LIN {X 0,Y 522.426,Z 691.44,A -85,B 0,C 180,E1 4711.435,E2 4711.435} C_VEL
LIN {X 0,Y 522.387,Z 691.44,A -85,B 0,C 180,E1 4717.482,E2 4717.482} C_VEL
LIN {X 0,Y 522.255,Z 691.44,A -85,B 0,C 180,E1 4723.549,E2 4723.549} C_VEL
LIN {X 0,Y 522.445,Z 691.44,A -85,B 0,C 180,E1 4730.119,E2 4730.119} C_VEL
LIN {X 0,Y 522.544,Z 692.414,A -85,B 0,C 180,E1 4730.325,E2 4730.325} C_VEL
LIN {X 0,Y 539.275,Z 726.671,A -85,B 0,C 180,E1 4732.514,E2 4732.514} C_VEL
LIN {X 0,Y 537.589,Z 764.271,A -85,B 0,C 180,E1 4733.74,E2 4733.74} C_VEL
LIN {X 0,Y 535.249,Z 801.949,A -85,B 0,C 180,E1 4735.545,E2 4735.545} C_VEL
LIN {X 0,Y 532.435,Z 840.351,A -85,B 0,C 180,E1 4738.098,E2 4738.098} C_VEL
LIN {X 0,Y 529.459,Z 877.291,A -85,B 0,C 180,E1 4741.38,E2 4741.38} C_VEL
LIN {X 0,Y 526.999,Z 909.325,A -85,B 0,C 180,E1 4745.105,E2 4745.105} C_VEL
LIN {X 0,Y 525.112,Z 937.42,A -85,B 0,C 180,E1 4749.358,E2 4749.358} C_VEL
LIN {X 0,Y 523.97,Z 958.909,A -85,B 0,C 180,E1 4753.636,E2 4753.636} C_VEL
LIN {X 0,Y 523.391,Z 974.577,A -85,B 0,C 180,E1 4757.893,E2 4757.893} C_VEL
LIN {X 0,Y 523.168,Z 984.427,A -85,B 0,C 180,E1 4761.68,E2 4761.68} C_VEL
LIN {X 0,Y 523.113,Z 989.961,A -85,B 0,C 180,E1 4765.018,E2 4765.018} C_VEL
LIN {X 0,Y 523.072,Z 992.674,A -85,B 0,C 180,E1 4768.341,E2 4768.341} C_VEL
LIN {X 0,Y 523.125,Z 992.634,A -85,B 0,C 180,E1 4771.658,E2 4771.658} C_VEL
LIN {X 0,Y 523.173,Z 988.638,A -85,B 0,C 180,E1 4775.813,E2 4775.813} C_VEL
LIN {X 0,Y 523.346,Z 980.316,A -85,B 0,C 180,E1 4779.996,E2 4779.996} C_VEL
LIN {X 0,Y 523.726,Z 965.346,A -85,B 0,C 180,E1 4784.698,E2 4784.698} C_VEL
LIN {X 0,Y 524.624,Z 945.078,A -85,B 0,C 180,E1 4789.164,E2 4789.164} C_VEL
LIN {X 0,Y 526.306,Z 918.749,A -85,B 0,C 180,E1 4793.507,E2 4793.507} C_VEL
LIN {X 0,Y 528.671,Z 887.696,A -85,B 0,C 180,E1 4797.423,E2 4797.423} C_VEL
LIN {X 0,Y 531.474,Z 852.279,A -85,B 0,C 180,E1 4800.85,E2 4800.85} C_VEL
LIN {X 0,Y 534.394,Z 814.101,A -85,B 0,C 180,E1 4803.642,E2 4803.642} C_VEL
LIN {X 0,Y 537.05,Z 773.839,A -85,B 0,C 180,E1 4805.776,E2 4805.776} C_VEL
LIN {X 0,Y 539,Z 734.912,A -85,B 0,C 180,E1 4807.168,E2 4807.168} C_VEL
LIN {X 0,Y 538.832,Z 725.059,A -85,B 0,C 180,E1 4807.474,E2 4807.474} C_VEL
LIN {X 0,Y 522.37,Z 692.689,A -85,B 0,C 180,E1 4809.596,E2 4809.596} C_VEL
LIN {X 0,Y 522.274,Z 691.44,A -85,B 0,C 180,E1 4809.626,E2 4809.626} C_VEL
LIN {X 0,Y 522.4,Z 691.44,A -85,B 0,C 180,E1 4815.938,E2 4815.938} C_VEL
LIN {X 0,Y 522.319,Z 691.44,A -85,B 0,C 180,E1 4821.505,E2 4821.505} C_VEL
LIN {X 0,Y 522.347,Z 691.44,A -85,B 0,C 180,E1 4827.203,E2 4827.203} C_VEL
LIN {X 0,Y 522.46,Z 691.44,A -85,B 0,C 180,E1 4832.384,E2 4832.384} C_VEL
LIN {X 0,Y 522.611,Z 691.44,A -85,B 0,C 180,E1 4837.985,E2 4837.985} C_VEL
LIN {X 0,Y 522.696,Z 691.44,A -85,B 0,C 180,E1 4843.169,E2 4843.169} C_VEL
LIN {X 0,Y 522.745,Z 691.44,A -85,B 0,C 180,E1 4848.308,E2 4848.308} C_VEL
LIN {X 0,Y 522.774,Z 691.44,A -85,B 0,C 180,E1 4853.352,E2 4853.352} C_VEL
LIN {X 0,Y 522.845,Z 691.44,A -85,B 0,C 180,E1 4858.345,E2 4858.345} C_VEL
LIN {X 0,Y 522.824,Z 691.44,A -85,B 0,C 180,E1 4863.324,E2 4863.324} C_VEL
LIN {X 0,Y 522.696,Z 691.44,A -85,B 0,C 180,E1 4868.331,E2 4868.331} C_VEL
LIN {X 0,Y 522.66,Z 691.44,A -85,B 0,C 180,E1 4873.402,E2 4873.402} C_VEL
LIN {X 0,Y 522.58,Z 691.44,A -85,B 0,C 180,E1 4878.586,E2 4878.586} C_VEL
LIN {X 0,Y 522.567,Z 691.44,A -85,B 0,C 180,E1 4883.932,E2 4883.932} C_VEL
LIN {X 0,Y 522.359,Z 691.44,A -85,B 0,C 180,E1 4889.593,E2 4889.593} C_VEL
LIN {X 0,Y 522.321,Z 691.44,A -85,B 0,C 180,E1 4892.498,E2 4892.498} C_VEL
LIN {X 0,Y 519.868,Z 691.44,A -85,B 0,C 180,E1 4893.912,E2 4893.912} C_VEL
LIN {X 0,Y 514.507,Z 691.44,A -85,B 0,C 180,E1 4896.031,E2 4896.031} C_VEL
LIN {X 0,Y 514.405,Z 691.44,A -85,B 0,C 180,E1 4896.276,E2 4896.276} C_VEL
LIN {X 0,Y 514.452,Z 691.44,A -85,B 0,C 180,E1 4902.601,E2 4902.601} C_VEL
LIN {X 0,Y 514.39,Z 691.44,A -85,B 0,C 180,E1 4909.063,E2 4909.063} C_VEL
LIN {X 0,Y 516.656,Z 696.972,A -85,B 0,C 180,E1 4909.378,E2 4909.378} C_VEL
LIN {X 0,Y 533.601,Z 728.662,A -85,B 0,C 180,E1 4911.452,E2 4911.452} C_VEL
LIN {X 0,Y 532.248,Z 772.885,A -85,B 0,C 180,E1 4912.494,E2 4912.494} C_VEL
LIN {X 0,Y 529.856,Z 813.695,A -85,B 0,C 180,E1 4914.129,E2 4914.129} C_VEL
LIN {X 0,Y 526.866,Z 853.448,A -85,B 0,C 180,E1 4916.444,E2 4916.444} C_VEL
LIN {X 0,Y 523.9,Z 889.133,A -85,B 0,C 180,E1 4919.257,E2 4919.257} C_VEL
LIN {X 0,Y 521.019,Z 921.486,A -85,B 0,C 180,E1 4922.555,E2 4922.555} C_VEL
LIN {X 0,Y 518.699,Z 950.198,A -85,B 0,C 180,E1 4926.305,E2 4926.305} C_VEL
LIN {X 0,Y 516.878,Z 975.351,A -85,B 0,C 180,E1 4930.546,E2 4930.546} C_VEL
LIN {X 0,Y 515.909,Z 995.049,A -85,B 0,C 180,E1 4934.952,E2 4934.952} C_VEL
LIN {X 0,Y 515.398,Z 1009.438,A -85,B 0,C 180,E1 4939.475,E2 4939.475} C_VEL
LIN {X 0,Y 515.274,Z 1017.479,A -85,B 0,C 180,E1 4943.25,E2 4943.25} C_VEL
LIN {X 0,Y 515.21,Z 1022.223,A -85,B 0,C 180,E1 4947.588,E2 4947.588} C_VEL
LIN {X 0,Y 515.151,Z 1022.657,A -85,B 0,C 180,E1 4951.685,E2 4951.685} C_VEL
LIN {X 0,Y 515.278,Z 1018.703,A -85,B 0,C 180,E1 4955.903,E2 4955.903} C_VEL
LIN {X 0,Y 515.502,Z 1010.436,A -85,B 0,C 180,E1 4960.15,E2 4960.15} C_VEL
LIN {X 0,Y 515.962,Z 995.944,A -85,B 0,C 180,E1 4964.803,E2 4964.803} C_VEL
LIN {X 0,Y 516.915,Z 975.395,A -85,B 0,C 180,E1 4969.443,E2 4969.443} C_VEL
LIN {X 0,Y 518.818,Z 949.033,A -85,B 0,C 180,E1 4973.869,E2 4973.869} C_VEL
LIN {X 0,Y 521.438,Z 917.371,A -85,B 0,C 180,E1 4977.919,E2 4977.919} C_VEL
LIN {X 0,Y 524.469,Z 882.798,A -85,B 0,C 180,E1 4981.308,E2 4981.308} C_VEL
LIN {X 0,Y 527.597,Z 844.909,A -85,B 0,C 180,E1 4984.124,E2 4984.124} C_VEL
LIN {X 0,Y 530.493,Z 804.797,A -85,B 0,C 180,E1 4986.284,E2 4986.284} C_VEL
LIN {X 0,Y 532.713,Z 762.573,A -85,B 0,C 180,E1 4987.804,E2 4987.804} C_VEL
LIN {X 0,Y 533.345,Z 728.122,A -85,B 0,C 180,E1 4988.579,E2 4988.579} C_VEL
LIN {X 0,Y 514.534,Z 692.798,A -85,B 0,C 180,E1 4990.898,E2 4990.898} C_VEL
LIN {X 0,Y 514.426,Z 691.44,A -85,B 0,C 180,E1 4991.055,E2 4991.055} C_VEL
LIN {X 0,Y 514.439,Z 691.44,A -85,B 0,C 180,E1 4997.398,E2 4997.398} C_VEL
LIN {X 0,Y 514.454,Z 691.44,A -85,B 0,C 180,E1 5002.621,E2 5002.621} C_VEL
LIN {X 0,Y 514.454,Z 691.44,A -85,B 0,C 180,E1 5008.595,E2 5008.595} C_VEL
LIN {X 0,Y 514.559,Z 691.44,A -85,B 0,C 180,E1 5013.808,E2 5013.808} C_VEL
LIN {X 0,Y 514.675,Z 691.44,A -85,B 0,C 180,E1 5019.327,E2 5019.327} C_VEL
LIN {X 0,Y 514.565,Z 691.44,A -85,B 0,C 180,E1 5024.642,E2 5024.642} C_VEL
LIN {X 0,Y 514.737,Z 691.44,A -85,B 0,C 180,E1 5029.832,E2 5029.832} C_VEL
LIN {X 0,Y 514.959,Z 691.44,A -85,B 0,C 180,E1 5034.936,E2 5034.936} C_VEL
LIN {X 0,Y 515.019,Z 691.44,A -85,B 0,C 180,E1 5039.996,E2 5039.996} C_VEL
LIN {X 0,Y 514.944,Z 691.44,A -85,B 0,C 180,E1 5045.056,E2 5045.056} C_VEL
LIN {X 0,Y 514.872,Z 691.44,A -85,B 0,C 180,E1 5050.157,E2 5050.157} C_VEL
LIN {X 0,Y 514.778,Z 691.44,A -85,B 0,C 180,E1 5055.343,E2 5055.343} C_VEL
LIN {X 0,Y 514.675,Z 691.44,A -85,B 0,C 180,E1 5060.665,E2 5060.665} C_VEL
LIN {X 0,Y 514.55,Z 691.44,A -85,B 0,C 180,E1 5066.184,E2 5066.184} C_VEL
LIN {X 0,Y 514.549,Z 691.44,A -85,B 0,C 180,E1 5071.973,E2 5071.973} C_VEL
LIN {X 0,Y 514.472,Z 691.44,A -85,B 0,C 180,E1 5078.161,E2 5078.161} C_VEL
LIN {X 0,Y 514.337,Z 691.44,A -85,B 0,C 180,E1 5082.613,E2 5082.613} C_VEL
LIN {X 0,Y 514.486,Z 691.44,A -85,B 0,C 180,E1 5089.553,E2 5089.553} C_VEL
LIN {X 0,Y 518.78,Z 700.928,A -85,B 0,C 180,E1 5090.135,E2 5090.135} C_VEL
LIN {X 0,Y 532.868,Z 728.329,A -85,B 0,C 180,E1 5092.028,E2 5092.028} C_VEL
LIN {X 0,Y 530.904,Z 768.275,A -85,B 0,C 180,E1 5093.392,E2 5093.392} C_VEL
LIN {X 0,Y 528.322,Z 805.367,A -85,B 0,C 180,E1 5095.254,E2 5095.254} C_VEL
LIN {X 0,Y 525.28,Z 843.001,A -85,B 0,C 180,E1 5097.842,E2 5097.842} C_VEL
LIN {X 0,Y 522.172,Z 878.329,A -85,B 0,C 180,E1 5101.061,E2 5101.061} C_VEL
LIN {X 0,Y 519.593,Z 909.281,A -85,B 0,C 180,E1 5104.719,E2 5104.719} C_VEL
LIN {X 0,Y 517.486,Z 937.186,A -85,B 0,C 180,E1 5108.997,E2 5108.997} C_VEL
LIN {X 0,Y 516.17,Z 958.905,A -85,B 0,C 180,E1 5113.381,E2 5113.381} C_VEL
LIN {X 0,Y 515.535,Z 974.574,A -85,B 0,C 180,E1 5117.706,E2 5117.706} C_VEL
LIN {X 0,Y 515.281,Z 984.426,A -85,B 0,C 180,E1 5121.551,E2 5121.551} C_VEL
LIN {X 0,Y 515.228,Z 989.96,A -85,B 0,C 180,E1 5124.942,E2 5124.942} C_VEL
LIN {X 0,Y 515.171,Z 992.674,A -85,B 0,C 180,E1 5128.316,E2 5128.316} C_VEL
LIN {X 0,Y 515.143,Z 992.185,A -85,B 0,C 180,E1 5132.429,E2 5132.429} C_VEL
LIN {X 0,Y 515.253,Z 987.399,A -85,B 0,C 180,E1 5136.75,E2 5136.75} C_VEL
LIN {X 0,Y 515.468,Z 977.399,A -85,B 0,C 180,E1 5141.237,E2 5141.237} C_VEL
LIN {X 0,Y 515.923,Z 963.805,A -85,B 0,C 180,E1 5145.315,E2 5145.315} C_VEL
LIN {X 0,Y 516.943,Z 943.977,A -85,B 0,C 180,E1 5149.679,E2 5149.679} C_VEL
LIN {X 0,Y 518.796,Z 918.754,A -85,B 0,C 180,E1 5153.869,E2 5153.869} C_VEL
LIN {X 0,Y 521.415,Z 887.703,A -85,B 0,C 180,E1 5157.838,E2 5157.838} C_VEL
LIN {X 0,Y 524.471,Z 852.291,A -85,B 0,C 180,E1 5161.308,E2 5161.308} C_VEL
LIN {X 0,Y 527.69,Z 813.795,A -85,B 0,C 180,E1 5164.149,E2 5164.149} C_VEL
LIN {X 0,Y 530.577,Z 773.856,A -85,B 0,C 180,E1 5166.282,E2 5166.282} C_VEL
LIN {X 0,Y 532.746,Z 734.504,A -85,B 0,C 180,E1 5167.693,E2 5167.693} C_VEL
LIN {X 0,Y 532.192,Z 727.448,A -85,B 0,C 180,E1 5167.962,E2 5167.962} C_VEL
LIN {X 0,Y 514.479,Z 692.831,A -85,B 0,C 180,E1 5170.331,E2 5170.331} C_VEL
LIN {X 0,Y 514.347,Z 691.44,A -85,B 0,C 180,E1 5170.542,E2 5170.542} C_VEL
LIN {X 0,Y 514.415,Z 691.44,A -85,B 0,C 180,E1 5175.071,E2 5175.071} C_VEL
LIN {X 0,Y 514.472,Z 691.44,A -85,B 0,C 180,E1 5179.922,E2 5179.922} C_VEL
LIN {X 0,Y 514.359,Z 691.44,A -85,B 0,C 180,E1 5186.004,E2 5186.004} C_VEL
LIN {X 0,Y 514.501,Z 691.44,A -85,B 0,C 180,E1 5191.987,E2 5191.987} C_VEL
LIN {X 0,Y 514.647,Z 691.44,A -85,B 0,C 180,E1 5197.522,E2 5197.522} C_VEL
LIN {X 0,Y 514.776,Z 691.44,A -85,B 0,C 180,E1 5202.902,E2 5202.902} C_VEL
LIN {X 0,Y 514.832,Z 691.44,A -85,B 0,C 180,E1 5208.126,E2 5208.126} C_VEL
LIN {X 0,Y 514.864,Z 691.44,A -85,B 0,C 180,E1 5213.25,E2 5213.25} C_VEL
LIN {X 0,Y 514.956,Z 691.44,A -85,B 0,C 180,E1 5218.526,E2 5218.526} C_VEL
LIN {X 0,Y 514.92,Z 691.44,A -85,B 0,C 180,E1 5223.375,E2 5223.375} C_VEL
LIN {X 0,Y 514.782,Z 691.44,A -85,B 0,C 180,E1 5228.46,E2 5228.46} C_VEL
LIN {X 0,Y 514.733,Z 691.44,A -85,B 0,C 180,E1 5233.907,E2 5233.907} C_VEL
LIN {X 0,Y 514.621,Z 691.44,A -85,B 0,C 180,E1 5239.699,E2 5239.699} C_VEL
LIN {X 0,Y 514.641,Z 691.44,A -85,B 0,C 180,E1 5244.324,E2 5244.324} C_VEL
LIN {X 0,Y 514.421,Z 691.44,A -85,B 0,C 180,E1 5250.024,E2 5250.024} C_VEL
LIN {X 0,Y 514.405,Z 691.44,A -85,B 0,C 180,E1 5256.276,E2 5256.276} C_VEL
LIN {X 0,Y 513.115,Z 691.44,A -85,B 0,C 180,E1 5257.239,E2 5257.239} C_VEL
LIN {X 0,Y 506.485,Z 691.44,A -85,B 0,C 180,E1 5259.86,E2 5259.86} C_VEL
LIN {X 0,Y 506.394,Z 691.44,A -85,B 0,C 180,E1 5260.108,E2 5260.108} C_VEL
LIN {X 0,Y 506.412,Z 691.44,A -85,B 0,C 180,E1 5265.851,E2 5265.851} C_VEL
LIN {X 0,Y 506.521,Z 691.58,A -85,B 0,C 180,E1 5268.297,E2 5268.297} C_VEL
LIN {X 0,Y 510.766,Z 700.951,A -85,B 0,C 180,E1 5268.886,E2 5268.886} C_VEL
LIN {X 0,Y 527.479,Z 731.737,A -85,B 0,C 180,E1 5270.981,E2 5270.981} C_VEL
LIN {X 0,Y 525.902,Z 773.975,A -85,B 0,C 180,E1 5272,E2 5272} C_VEL
LIN {X 0,Y 523.228,Z 816.041,A -85,B 0,C 180,E1 5273.727,E2 5273.727} C_VEL
LIN {X 0,Y 519.776,Z 857.497,A -85,B 0,C 180,E1 5276.226,E2 5276.226} C_VEL
LIN {X 0,Y 516.312,Z 895.403,A -85,B 0,C 180,E1 5279.368,E2 5279.368} C_VEL
LIN {X 0,Y 513.008,Z 929.647,A -85,B 0,C 180,E1 5283.115,E2 5283.115} C_VEL
LIN {X 0,Y 510.483,Z 959.035,A -85,B 0,C 180,E1 5287.321,E2 5287.321} C_VEL
LIN {X 0,Y 508.819,Z 982.147,A -85,B 0,C 180,E1 5291.635,E2 5291.635} C_VEL
LIN {X 0,Y 507.923,Z 1000.301,A -85,B 0,C 180,E1 5296.204,E2 5296.204} C_VEL
LIN {X 0,Y 507.526,Z 1012.606,A -85,B 0,C 180,E1 5300.646,E2 5300.646} C_VEL
LIN {X 0,Y 507.424,Z 1019.905,A -85,B 0,C 180,E1 5304.865,E2 5304.865} C_VEL
LIN {X 0,Y 507.396,Z 1022.657,A -85,B 0,C 180,E1 5308.29,E2 5308.29} C_VEL
LIN {X 0,Y 507.319,Z 1021.627,A -85,B 0,C 180,E1 5313.422,E2 5313.422} C_VEL
LIN {X 0,Y 507.443,Z 1015.917,A -85,B 0,C 180,E1 5317.717,E2 5317.717} C_VEL
LIN {X 0,Y 507.636,Z 1005.771,A -85,B 0,C 180,E1 5322.051,E2 5322.051} C_VEL
LIN {X 0,Y 508.318,Z 990.49,A -85,B 0,C 180,E1 5326.438,E2 5326.438} C_VEL
LIN {X 0,Y 509.72,Z 969.378,A -85,B 0,C 180,E1 5330.883,E2 5330.883} C_VEL
LIN {X 0,Y 511.785,Z 943.259,A -85,B 0,C 180,E1 5335.069,E2 5335.069} C_VEL
LIN {X 0,Y 514.543,Z 913.188,A -85,B 0,C 180,E1 5338.806,E2 5338.806} C_VEL
LIN {X 0,Y 517.862,Z 878.743,A -85,B 0,C 180,E1 5342.117,E2 5342.117} C_VEL
LIN {X 0,Y 521.115,Z 842.642,A -85,B 0,C 180,E1 5344.764,E2 5344.764} C_VEL
LIN {X 0,Y 524.261,Z 802.755,A -85,B 0,C 180,E1 5346.894,E2 5346.894} C_VEL
LIN {X 0,Y 526.437,Z 762.992,A -85,B 0,C 180,E1 5348.322,E2 5348.322} C_VEL
LIN {X 0,Y 526.991,Z 730.718,A -85,B 0,C 180,E1 5349.082,E2 5349.082} C_VEL
LIN {X 0,Y 506.659,Z 692.982,A -85,B 0,C 180,E1 5351.664,E2 5351.664} C_VEL
LIN {X 0,Y 506.519,Z 691.44,A -85,B 0,C 180,E1 5351.811,E2 5351.811} C_VEL
LIN {X 0,Y 506.485,Z 691.44,A -85,B 0,C 180,E1 5358.362,E2 5358.362} C_VEL
LIN {X 0,Y 506.537,Z 691.44,A -85,B 0,C 180,E1 5363.81,E2 5363.81} C_VEL
LIN {X 0,Y 506.517,Z 691.44,A -85,B 0,C 180,E1 5370.098,E2 5370.098} C_VEL
LIN {X 0,Y 506.639,Z 691.44,A -85,B 0,C 180,E1 5375.266,E2 5375.266} C_VEL
LIN {X 0,Y 506.813,Z 691.44,A -85,B 0,C 180,E1 5380.813,E2 5380.813} C_VEL
LIN {X 0,Y 506.617,Z 691.44,A -85,B 0,C 180,E1 5386.165,E2 5386.165} C_VEL
LIN {X 0,Y 506.849,Z 691.44,A -85,B 0,C 180,E1 5391.407,E2 5391.407} C_VEL
LIN {X 0,Y 507.02,Z 691.44,A -85,B 0,C 180,E1 5396.572,E2 5396.572} C_VEL
LIN {X 0,Y 507.072,Z 691.44,A -85,B 0,C 180,E1 5401.707,E2 5401.707} C_VEL
LIN {X 0,Y 506.955,Z 691.44,A -85,B 0,C 180,E1 5406.856,E2 5406.856} C_VEL
LIN {X 0,Y 506.856,Z 691.44,A -85,B 0,C 180,E1 5412.064,E2 5412.064} C_VEL
LIN {X 0,Y 506.807,Z 691.44,A -85,B 0,C 180,E1 5417.376,E2 5417.376} C_VEL
LIN {X 0,Y 506.713,Z 691.44,A -85,B 0,C 180,E1 5422.85,E2 5422.85} C_VEL
LIN {X 0,Y 506.544,Z 691.44,A -85,B 0,C 180,E1 5428.562,E2 5428.562} C_VEL
LIN {X 0,Y 506.601,Z 691.44,A -85,B 0,C 180,E1 5434.59,E2 5434.59} C_VEL
LIN {X 0,Y 506.421,Z 691.44,A -85,B 0,C 180,E1 5441.116,E2 5441.116} C_VEL
LIN {X 0,Y 506.374,Z 691.44,A -85,B 0,C 180,E1 5446.55,E2 5446.55} C_VEL
LIN {X 0,Y 506.584,Z 691.44,A -85,B 0,C 180,E1 5448.757,E2 5448.757} C_VEL
LIN {X 0,Y 511.353,Z 701.712,A -85,B 0,C 180,E1 5449.447,E2 5449.447} C_VEL
LIN {X 0,Y 526.49,Z 731.264,A -85,B 0,C 180,E1 5451.58,E2 5451.58} C_VEL
LIN {X 0,Y 524.243,Z 772.496,A -85,B 0,C 180,E1 5453.047,E2 5453.047} C_VEL
LIN {X 0,Y 521.209,Z 811.429,A -85,B 0,C 180,E1 5455.116,E2 5455.116} C_VEL
LIN {X 0,Y 517.884,Z 848.298,A -85,B 0,C 180,E1 5457.8,E2 5457.8} C_VEL
LIN {X 0,Y 514.557,Z 882.537,A -85,B 0,C 180,E1 5461.076,E2 5461.076} C_VEL
LIN {X 0,Y 511.836,Z 912.444,A -85,B 0,C 180,E1 5464.77,E2 5464.77} C_VEL
LIN {X 0,Y 509.755,Z 938.401,A -85,B 0,C 180,E1 5468.891,E2 5468.891} C_VEL
LIN {X 0,Y 508.391,Z 958.902,A -85,B 0,C 180,E1 5473.119,E2 5473.119} C_VEL
LIN {X 0,Y 507.692,Z 974.571,A -85,B 0,C 180,E1 5477.513,E2 5477.513} C_VEL
LIN {X 0,Y 507.391,Z 984.424,A -85,B 0,C 180,E1 5481.419,E2 5481.419} C_VEL
LIN {X 0,Y 507.331,Z 989.959,A -85,B 0,C 180,E1 5484.863,E2 5484.863} C_VEL
LIN {X 0,Y 507.291,Z 992.674,A -85,B 0,C 180,E1 5488.289,E2 5488.289} C_VEL
LIN {X 0,Y 507.334,Z 992.635,A -85,B 0,C 180,E1 5491.71,E2 5491.71} C_VEL
LIN {X 0,Y 507.375,Z 988.64,A -85,B 0,C 180,E1 5495.995,E2 5495.995} C_VEL
LIN {X 0,Y 507.59,Z 979.171,A -85,B 0,C 180,E1 5500.744,E2 5500.744} C_VEL
LIN {X 0,Y 508.044,Z 965.517,A -85,B 0,C 180,E1 5505.116,E2 5505.116} C_VEL
LIN {X 0,Y 509.156,Z 945.376,A -85,B 0,C 180,E1 5509.711,E2 5509.711} C_VEL
LIN {X 0,Y 511.113,Z 920.579,A -85,B 0,C 180,E1 5513.963,E2 5513.963} C_VEL
LIN {X 0,Y 513.822,Z 890.873,A -85,B 0,C 180,E1 5517.894,E2 5517.894} C_VEL
LIN {X 0,Y 517.003,Z 857.416,A -85,B 0,C 180,E1 5521.32,E2 5521.32} C_VEL
LIN {X 0,Y 520.294,Z 822.156,A -85,B 0,C 180,E1 5524.088,E2 5524.088} C_VEL
LIN {X 0,Y 523.368,Z 783.668,A -85,B 0,C 180,E1 5526.343,E2 5526.343} C_VEL
LIN {X 0,Y 526.016,Z 743.231,A -85,B 0,C 180,E1 5527.972,E2 5527.972} C_VEL
LIN {X 0,Y 526.121,Z 731.045,A -85,B 0,C 180,E1 5528.369,E2 5528.369} C_VEL
LIN {X 0,Y 506.531,Z 692.262,A -85,B 0,C 180,E1 5531.117,E2 5531.117} C_VEL
LIN {X 0,Y 506.507,Z 691.44,A -85,B 0,C 180,E1 5531.657,E2 5531.657} C_VEL
LIN {X 0,Y 506.483,Z 691.44,A -85,B 0,C 180,E1 5538.361,E2 5538.361} C_VEL
LIN {X 0,Y 506.5,Z 691.44,A -85,B 0,C 180,E1 5543.814,E2 5543.814} C_VEL
LIN {X 0,Y 506.528,Z 691.44,A -85,B 0,C 180,E1 5550.094,E2 5550.094} C_VEL
LIN {X 0,Y 506.677,Z 691.44,A -85,B 0,C 180,E1 5555.277,E2 5555.277} C_VEL
LIN {X 0,Y 506.822,Z 691.44,A -85,B 0,C 180,E1 5560.822,E2 5560.822} C_VEL
LIN {X 0,Y 506.985,Z 691.44,A -85,B 0,C 180,E1 5566.184,E2 5566.184} C_VEL
LIN {X 0,Y 507.008,Z 691.44,A -85,B 0,C 180,E1 5571.418,E2 5571.418} C_VEL
LIN {X 0,Y 507.178,Z 691.44,A -85,B 0,C 180,E1 5576.582,E2 5576.582} C_VEL
LIN {X 0,Y 507.295,Z 691.44,A -85,B 0,C 180,E1 5581.714,E2 5581.714} C_VEL
LIN {X 0,Y 507.062,Z 691.44,A -85,B 0,C 180,E1 5586.863,E2 5586.863} C_VEL
LIN {X 0,Y 506.869,Z 691.44,A -85,B 0,C 180,E1 5592.072,E2 5592.072} C_VEL
LIN {X 0,Y 506.779,Z 691.44,A -85,B 0,C 180,E1 5597.385,E2 5597.385} C_VEL
LIN {X 0,Y 506.729,Z 691.44,A -85,B 0,C 180,E1 5602.858,E2 5602.858} C_VEL
LIN {X 0,Y 506.529,Z 691.44,A -85,B 0,C 180,E1 5608.572,E2 5608.572} C_VEL
LIN {X 0,Y 506.47,Z 691.44,A -85,B 0,C 180,E1 5614.611,E2 5614.611} C_VEL
LIN {X 0,Y 506.394,Z 691.44,A -85,B 0,C 180,E1 5620.108,E2 5620.108} C_VEL
LIN {X 0,Y 503.895,Z 691.44,A -85,B 0,C 180,E1 5621.569,E2 5621.569} C_VEL
LIN {X 0,Y 498.621,Z 691.44,A -85,B 0,C 180,E1 5623.758,E2 5623.758} C_VEL
LIN {X 0,Y 498.534,Z 691.44,A -85,B 0,C 180,E1 5624.011,E2 5624.011} C_VEL
LIN {X 0,Y 498.582,Z 691.44,A -85,B 0,C 180,E1 5627.457,E2 5627.457} C_VEL
LIN {X 0,Y 503.054,Z 701.159,A -85,B 0,C 180,E1 5628.126,E2 5628.126} C_VEL
LIN {X 0,Y 521.229,Z 734.453,A -85,B 0,C 180,E1 5630.479,E2 5630.479} C_VEL
LIN {X 0,Y 519.57,Z 775.534,A -85,B 0,C 180,E1 5631.516,E2 5631.516} C_VEL
LIN {X 0,Y 516.672,Z 817.16,A -85,B 0,C 180,E1 5633.256,E2 5633.256} C_VEL
LIN {X 0,Y 512.985,Z 858.207,A -85,B 0,C 180,E1 5635.775,E2 5635.775} C_VEL
LIN {X 0,Y 509.262,Z 895.435,A -85,B 0,C 180,E1 5638.901,E2 5638.901} C_VEL
LIN {X 0,Y 505.79,Z 928.839,A -85,B 0,C 180,E1 5642.589,E2 5642.589} C_VEL
LIN {X 0,Y 502.862,Z 959.037,A -85,B 0,C 180,E1 5646.957,E2 5646.957} C_VEL
LIN {X 0,Y 501.01,Z 983.299,A -85,B 0,C 180,E1 5651.605,E2 5651.605} C_VEL
LIN {X 0,Y 500.042,Z 1001.746,A -85,B 0,C 180,E1 5656.429,E2 5656.429} C_VEL
LIN {X 0,Y 499.556,Z 1014.331,A -85,B 0,C 180,E1 5661.284,E2 5661.284} C_VEL
LIN {X 0,Y 499.53,Z 1019.905,A -85,B 0,C 180,E1 5664.783,E2 5664.783} C_VEL
LIN {X 0,Y 499.5,Z 1022.657,A -85,B 0,C 180,E1 5668.263,E2 5668.263} C_VEL
LIN {X 0,Y 499.413,Z 1021.627,A -85,B 0,C 180,E1 5673.477,E2 5673.477} C_VEL
LIN {X 0,Y 499.554,Z 1015.917,A -85,B 0,C 180,E1 5677.839,E2 5677.839} C_VEL
LIN {X 0,Y 499.774,Z 1005.77,A -85,B 0,C 180,E1 5682.244,E2 5682.244} C_VEL
LIN {X 0,Y 500.541,Z 990.491,A -85,B 0,C 180,E1 5686.701,E2 5686.701} C_VEL
LIN {X 0,Y 502.073,Z 969.379,A -85,B 0,C 180,E1 5691.216,E2 5691.216} C_VEL
LIN {X 0,Y 504.382,Z 943.018,A -85,B 0,C 180,E1 5695.498,E2 5695.498} C_VEL
LIN {X 0,Y 507.324,Z 913.665,A -85,B 0,C 180,E1 5699.199,E2 5699.199} C_VEL
LIN {X 0,Y 510.819,Z 880.199,A -85,B 0,C 180,E1 5702.482,E2 5702.482} C_VEL
LIN {X 0,Y 514.483,Z 842.657,A -85,B 0,C 180,E1 5705.278,E2 5705.278} C_VEL
LIN {X 0,Y 517.913,Z 802.357,A -85,B 0,C 180,E1 5707.443,E2 5707.443} C_VEL
LIN {X 0,Y 520.361,Z 761.523,A -85,B 0,C 180,E1 5708.902,E2 5708.902} C_VEL
LIN {X 0,Y 520.917,Z 733.875,A -85,B 0,C 180,E1 5709.561,E2 5709.561} C_VEL
LIN {X 0,Y 498.647,Z 692.273,A -85,B 0,C 180,E1 5712.494,E2 5712.494} C_VEL
LIN {X 0,Y 498.552,Z 691.44,A -85,B 0,C 180,E1 5713.21,E2 5713.21} C_VEL
LIN {X 0,Y 498.514,Z 691.44,A -85,B 0,C 180,E1 5719.403,E2 5719.403} C_VEL
LIN {X 0,Y 498.573,Z 691.44,A -85,B 0,C 180,E1 5725.08,E2 5725.08} C_VEL
LIN {X 0,Y 498.583,Z 691.44,A -85,B 0,C 180,E1 5731.723,E2 5731.723} C_VEL
LIN {X 0,Y 498.759,Z 691.44,A -85,B 0,C 180,E1 5736.755,E2 5736.755} C_VEL
LIN {X 0,Y 498.876,Z 691.44,A -85,B 0,C 180,E1 5742.33,E2 5742.33} C_VEL
LIN {X 0,Y 498.771,Z 691.44,A -85,B 0,C 180,E1 5747.729,E2 5747.729} C_VEL
LIN {X 0,Y 499.133,Z 691.44,A -85,B 0,C 180,E1 5753.027,E2 5753.027} C_VEL
LIN {X 0,Y 499.38,Z 691.44,A -85,B 0,C 180,E1 5758.259,E2 5758.259} C_VEL
LIN {X 0,Y 499.259,Z 691.44,A -85,B 0,C 180,E1 5763.473,E2 5763.473} C_VEL
LIN {X 0,Y 499.072,Z 691.44,A -85,B 0,C 180,E1 5768.719,E2 5768.719} C_VEL
LIN {X 0,Y 498.969,Z 691.44,A -85,B 0,C 180,E1 5774.043,E2 5774.043} C_VEL
LIN {X 0,Y 498.825,Z 691.44,A -85,B 0,C 180,E1 5779.788,E2 5779.788} C_VEL
LIN {X 0,Y 498.728,Z 691.44,A -85,B 0,C 180,E1 5785.144,E2 5785.144} C_VEL
LIN {X 0,Y 498.626,Z 691.44,A -85,B 0,C 180,E1 5791.763,E2 5791.763} C_VEL
LIN {X 0,Y 498.561,Z 691.44,A -85,B 0,C 180,E1 5797.852,E2 5797.852} C_VEL
LIN {X 0,Y 498.431,Z 691.44,A -85,B 0,C 180,E1 5804.307,E2 5804.307} C_VEL
LIN {X 0,Y 498.577,Z 691.44,A -85,B 0,C 180,E1 5807.945,E2 5807.945} C_VEL
LIN {X 0,Y 501.267,Z 697.296,A -85,B 0,C 180,E1 5808.355,E2 5808.355} C_VEL
LIN {X 0,Y 520.114,Z 734.342,A -85,B 0,C 180,E1 5811.126,E2 5811.126} C_VEL
LIN {X 0,Y 517.633,Z 775.019,A -85,B 0,C 180,E1 5812.631,E2 5812.631} C_VEL
LIN {X 0,Y 514.435,Z 813.313,A -85,B 0,C 180,E1 5814.718,E2 5814.718} C_VEL
LIN {X 0,Y 510.656,Z 851.969,A -85,B 0,C 180,E1 5817.623,E2 5817.623} C_VEL
LIN {X 0,Y 506.884,Z 887.913,A -85,B 0,C 180,E1 5821.225,E2 5821.225} C_VEL
LIN {X 0,Y 503.765,Z 919.734,A -85,B 0,C 180,E1 5825.438,E2 5825.438} C_VEL
LIN {X 0,Y 501.513,Z 945.589,A -85,B 0,C 180,E1 5829.929,E2 5829.929} C_VEL
LIN {X 0,Y 500.33,Z 965.611,A -85,B 0,C 180,E1 5834.581,E2 5834.581} C_VEL
LIN {X 0,Y 499.742,Z 980.552,A -85,B 0,C 180,E1 5839.526,E2 5839.526} C_VEL
LIN {X 0,Y 499.529,Z 988.765,A -85,B 0,C 180,E1 5843.91,E2 5843.91} C_VEL
LIN {X 0,Y 499.411,Z 992.673,A -85,B 0,C 180,E1 5848.262,E2 5848.262} C_VEL
LIN {X 0,Y 499.433,Z 992.636,A -85,B 0,C 180,E1 5851.737,E2 5851.737} C_VEL
LIN {X 0,Y 499.499,Z 988.641,A -85,B 0,C 180,E1 5856.09,E2 5856.09} C_VEL
LIN {X 0,Y 499.706,Z 980.32,A -85,B 0,C 180,E1 5860.474,E2 5860.474} C_VEL
LIN {X 0,Y 500.184,Z 966.655,A -85,B 0,C 180,E1 5865.031,E2 5865.031} C_VEL
LIN {X 0,Y 501.282,Z 948.378,A -85,B 0,C 180,E1 5869.405,E2 5869.405} C_VEL
LIN {X 0,Y 503.201,Z 925.226,A -85,B 0,C 180,E1 5873.615,E2 5873.615} C_VEL
LIN {X 0,Y 506.004,Z 896.865,A -85,B 0,C 180,E1 5877.606,E2 5877.606} C_VEL
LIN {X 0,Y 509.439,Z 863.725,A -85,B 0,C 180,E1 5881.215,E2 5881.215} C_VEL
LIN {X 0,Y 513.096,Z 827.618,A -85,B 0,C 180,E1 5884.22,E2 5884.22} C_VEL
LIN {X 0,Y 516.748,Z 786.229,A -85,B 0,C 180,E1 5886.747,E2 5886.747} C_VEL
LIN {X 0,Y 519.701,Z 744.166,A -85,B 0,C 180,E1 5888.483,E2 5888.483} C_VEL
LIN {X 0,Y 519.765,Z 734.009,A -85,B 0,C 180,E1 5888.826,E2 5888.826} C_VEL
LIN {X 0,Y 500.529,Z 696.592,A -85,B 0,C 180,E1 5891.644,E2 5891.644} C_VEL
LIN {X 0,Y 498.55,Z 691.44,A -85,B 0,C 180,E1 5892.061,E2 5892.061} C_VEL
LIN {X 0,Y 498.55,Z 691.44,A -85,B 0,C 180,E1 5898.09,E2 5898.09} C_VEL
LIN {X 0,Y 498.555,Z 691.44,A -85,B 0,C 180,E1 5904.77,E2 5904.77} C_VEL
LIN {X 0,Y 498.593,Z 691.44,A -85,B 0,C 180,E1 5910.94,E2 5910.94} C_VEL
LIN {X 0,Y 498.773,Z 691.44,A -85,B 0,C 180,E1 5916.765,E2 5916.765} C_VEL
LIN {X 0,Y 498.901,Z 691.44,A -85,B 0,C 180,E1 5922.34,E2 5922.34} C_VEL
LIN {X 0,Y 499.001,Z 691.44,A -85,B 0,C 180,E1 5927.743,E2 5927.743} C_VEL
LIN {X 0,Y 499.046,Z 691.44,A -85,B 0,C 180,E1 5933.035,E2 5933.035} C_VEL
LIN {X 0,Y 499.182,Z 691.44,A -85,B 0,C 180,E1 5938.266,E2 5938.266} C_VEL
LIN {X 0,Y 499.12,Z 691.44,A -85,B 0,C 180,E1 5943.482,E2 5943.482} C_VEL
LIN {X 0,Y 498.975,Z 691.44,A -85,B 0,C 180,E1 5948.73,E2 5948.73} C_VEL
LIN {X 0,Y 498.922,Z 691.44,A -85,B 0,C 180,E1 5954.053,E2 5954.053} C_VEL
LIN {X 0,Y 498.779,Z 691.44,A -85,B 0,C 180,E1 5959.776,E2 5959.776} C_VEL
LIN {X 0,Y 498.759,Z 691.44,A -85,B 0,C 180,E1 5965.151,E2 5965.151} C_VEL
LIN {X 0,Y 498.5,Z 691.44,A -85,B 0,C 180,E1 5971.741,E2 5971.741} C_VEL
LIN {X 0,Y 498.526,Z 691.44,A -85,B 0,C 180,E1 5977.848,E2 5977.848} C_VEL
LIN {X 0,Y 498.534,Z 691.44,A -85,B 0,C 180,E1 5984.011,E2 5984.011} C_VEL
LIN {X 0,Y 494.419,Z 691.225,A -85,B 0,C 180,E1 5985.297,E2 5985.297} C_VEL
LIN {X 0,Y 490.661,Z 691.355,A -85,B 0,C 180,E1 5986.428,E2 5986.428} C_VEL
LIN {X 0,Y 490.645,Z 691.452,A -85,B 0,C 180,E1 5986.601,E2 5986.601} C_VEL
LIN {X 0,Y 495.371,Z 701.46,A -85,B 0,C 180,E1 5987.338,E2 5987.338} C_VEL
LIN {X 0,Y 514.96,Z 737.17,A -85,B 0,C 180,E1 5989.963,E2 5989.963} C_VEL
LIN {X 0,Y 513.073,Z 779.161,A -85,B 0,C 180,E1 5991.088,E2 5991.088} C_VEL
LIN {X 0,Y 510.035,Z 819.606,A -85,B 0,C 180,E1 5992.85,E2 5992.85} C_VEL
LIN {X 0,Y 506.132,Z 859.584,A -85,B 0,C 180,E1 5995.363,E2 5995.363} C_VEL
LIN {X 0,Y 502.081,Z 896.882,A -85,B 0,C 180,E1 5998.565,E2 5998.565} C_VEL
LIN {X 0,Y 498.398,Z 929.579,A -85,B 0,C 180,E1 6002.251,E2 6002.251} C_VEL
LIN {X 0,Y 495.331,Z 959.039,A -85,B 0,C 180,E1 6006.586,E2 6006.586} C_VEL
LIN {X 0,Y 493.306,Z 982.847,A -85,B 0,C 180,E1 6011.2,E2 6011.2} C_VEL
LIN {X 0,Y 492.203,Z 1001.747,A -85,B 0,C 180,E1 6016.208,E2 6016.208} C_VEL
LIN {X 0,Y 491.674,Z 1014.331,A -85,B 0,C 180,E1 6021.143,E2 6021.143} C_VEL
LIN {X 0,Y 491.625,Z 1019.905,A -85,B 0,C 180,E1 6024.699,E2 6024.699} C_VEL
LIN {X 0,Y 491.594,Z 1022.657,A -85,B 0,C 180,E1 6028.235,E2 6028.235} C_VEL
LIN {X 0,Y 491.488,Z 1022.657,A -85,B 0,C 180,E1 6031.766,E2 6031.766} C_VEL
LIN {X 0,Y 491.621,Z 1018.703,A -85,B 0,C 180,E1 6036.188,E2 6036.188} C_VEL
LIN {X 0,Y 491.866,Z 1010.435,A -85,B 0,C 180,E1 6040.644,E2 6040.644} C_VEL
LIN {X 0,Y 492.466,Z 995.678,A -85,B 0,C 180,E1 6045.606,E2 6045.606} C_VEL
LIN {X 0,Y 493.802,Z 975.753,A -85,B 0,C 180,E1 6050.318,E2 6050.318} C_VEL
LIN {X 0,Y 496.192,Z 950.696,A -85,B 0,C 180,E1 6054.76,E2 6054.76} C_VEL
LIN {X 0,Y 499.353,Z 921.06,A -85,B 0,C 180,E1 6058.799,E2 6058.799} C_VEL
LIN {X 0,Y 503.125,Z 887.426,A -85,B 0,C 180,E1 6062.332,E2 6062.332} C_VEL
LIN {X 0,Y 506.966,Z 851.311,A -85,B 0,C 180,E1 6065.225,E2 6065.225} C_VEL
LIN {X 0,Y 510.6,Z 812.87,A -85,B 0,C 180,E1 6067.495,E2 6067.495} C_VEL
LIN {X 0,Y 513.488,Z 771.226,A -85,B 0,C 180,E1 6069.186,E2 6069.186} C_VEL
LIN {X 0,Y 514.897,Z 737.014,A -85,B 0,C 180,E1 6070.046,E2 6070.046} C_VEL
LIN {X 0,Y 490.815,Z 693.025,A -85,B 0,C 180,E1 6073.315,E2 6073.315} C_VEL
LIN {X 0,Y 490.634,Z 691.44,A -85,B 0,C 180,E1 6073.42,E2 6073.42} C_VEL
LIN {X 0,Y 490.605,Z 691.44,A -85,B 0,C 180,E1 6079.603,E2 6079.603} C_VEL
LIN {X 0,Y 490.617,Z 691.44,A -85,B 0,C 180,E1 6086.255,E2 6086.255} C_VEL
LIN {X 0,Y 490.689,Z 691.44,A -85,B 0,C 180,E1 6092.429,E2 6092.429} C_VEL
LIN {X 0,Y 490.87,Z 691.44,A -85,B 0,C 180,E1 6098.274,E2 6098.274} C_VEL
LIN {X 0,Y 490.867,Z 691.44,A -85,B 0,C 180,E1 6103.881,E2 6103.881} C_VEL
LIN {X 0,Y 490.983,Z 691.44,A -85,B 0,C 180,E1 6110.686,E2 6110.686} C_VEL
LIN {X 0,Y 491.218,Z 691.44,A -85,B 0,C 180,E1 6116.462,E2 6116.462} C_VEL
LIN {X 0,Y 491.285,Z 691.44,A -85,B 0,C 180,E1 6121.762,E2 6121.762} C_VEL
LIN {X 0,Y 491.133,Z 691.44,A -85,B 0,C 180,E1 6127.078,E2 6127.078} C_VEL
LIN {X 0,Y 491.03,Z 691.44,A -85,B 0,C 180,E1 6132.459,E2 6132.459} C_VEL
LIN {X 0,Y 490.952,Z 691.44,A -85,B 0,C 180,E1 6137.956,E2 6137.956} C_VEL
LIN {X 0,Y 490.829,Z 691.44,A -85,B 0,C 180,E1 6143.634,E2 6143.634} C_VEL
LIN {X 0,Y 490.665,Z 691.44,A -85,B 0,C 180,E1 6150.229,E2 6150.229} C_VEL
LIN {X 0,Y 490.661,Z 691.44,A -85,B 0,C 180,E1 6155.884,E2 6155.884} C_VEL
LIN {X 0,Y 490.549,Z 691.44,A -85,B 0,C 180,E1 6162.203,E2 6162.203} C_VEL
LIN {X 0,Y 490.601,Z 691.44,A -85,B 0,C 180,E1 6167.107,E2 6167.107} C_VEL
LIN {X 0,Y 492.937,Z 697.049,A -85,B 0,C 180,E1 6167.476,E2 6167.476} C_VEL
LIN {X 0,Y 511.652,Z 732.395,A -85,B 0,C 180,E1 6170.283,E2 6170.283} C_VEL
LIN {X 0,Y 513.7,Z 738.961,A -85,B 0,C 180,E1 6170.705,E2 6170.705} C_VEL
LIN {X 0,Y 510.881,Z 779.483,A -85,B 0,C 180,E1 6172.298,E2 6172.298} C_VEL
LIN {X 0,Y 507.486,Z 816.782,A -85,B 0,C 180,E1 6174.424,E2 6174.424} C_VEL
LIN {X 0,Y 503.504,Z 854.26,A -85,B 0,C 180,E1 6177.33,E2 6177.33} C_VEL
LIN {X 0,Y 499.692,Z 888.118,A -85,B 0,C 180,E1 6180.798,E2 6180.798} C_VEL
LIN {X 0,Y 496.307,Z 919.351,A -85,B 0,C 180,E1 6184.982,E2 6184.982} C_VEL
LIN {X 0,Y 493.949,Z 944.477,A -85,B 0,C 180,E1 6189.373,E2 6189.373} C_VEL
LIN {X 0,Y 492.536,Z 964.148,A -85,B 0,C 180,E1 6193.938,E2 6193.938} C_VEL
LIN {X 0,Y 491.873,Z 978.256,A -85,B 0,C 180,E1 6198.458,E2 6198.458} C_VEL
LIN {X 0,Y 491.618,Z 987.549,A -85,B 0,C 180,E1 6202.923,E2 6202.923} C_VEL
LIN {X 0,Y 491.587,Z 991.661,A -85,B 0,C 180,E1 6206.468,E2 6206.468} C_VEL
LIN {X 0,Y 491.527,Z 992.636,A -85,B 0,C 180,E1 6211.765,E2 6211.765} C_VEL
LIN {X 0,Y 491.61,Z 988.642,A -85,B 0,C 180,E1 6216.188,E2 6216.188} C_VEL
LIN {X 0,Y 491.838,Z 980.322,A -85,B 0,C 180,E1 6220.644,E2 6220.644} C_VEL
LIN {X 0,Y 492.413,Z 965.527,A -85,B 0,C 180,E1 6225.607,E2 6225.607} C_VEL
LIN {X 0,Y 493.81,Z 945.471,A -85,B 0,C 180,E1 6230.333,E2 6230.333} C_VEL
LIN {X 0,Y 496.209,Z 920.133,A -85,B 0,C 180,E1 6234.806,E2 6234.806} C_VEL
LIN {X 0,Y 499.608,Z 888.992,A -85,B 0,C 180,E1 6239.005,E2 6239.005} C_VEL
LIN {X 0,Y 503.671,Z 852.943,A -85,B 0,C 180,E1 6242.699,E2 6242.699} C_VEL
LIN {X 0,Y 507.793,Z 813.897,A -85,B 0,C 180,E1 6245.682,E2 6245.682} C_VEL
LIN {X 0,Y 511.496,Z 773.239,A -85,B 0,C 180,E1 6247.903,E2 6247.903} C_VEL
LIN {X 0,Y 513.453,Z 737.026,A -85,B 0,C 180,E1 6249.296,E2 6249.296} C_VEL
LIN {X 0,Y 494.942,Z 700.709,A -85,B 0,C 180,E1 6252.148,E2 6252.148} C_VEL
LIN {X 0,Y 490.694,Z 692.548,A -85,B 0,C 180,E1 6252.765,E2 6252.765} C_VEL
LIN {X 0,Y 490.628,Z 691.44,A -85,B 0,C 180,E1 6252.91,E2 6252.91} C_VEL
LIN {X 0,Y 490.657,Z 691.44,A -85,B 0,C 180,E1 6257.782,E2 6257.782} C_VEL
LIN {X 0,Y 490.564,Z 691.44,A -85,B 0,C 180,E1 6264.108,E2 6264.108} C_VEL
LIN {X 0,Y 490.618,Z 691.44,A -85,B 0,C 180,E1 6270.421,E2 6270.421} C_VEL
LIN {X 0,Y 490.846,Z 691.44,A -85,B 0,C 180,E1 6276.367,E2 6276.367} C_VEL
LIN {X 0,Y 490.979,Z 691.44,A -85,B 0,C 180,E1 6282.045,E2 6282.045} C_VEL
LIN {X 0,Y 491.093,Z 691.44,A -85,B 0,C 180,E1 6287.543,E2 6287.543} C_VEL
LIN {X 0,Y 491.137,Z 691.44,A -85,B 0,C 180,E1 6292.922,E2 6292.922} C_VEL
LIN {X 0,Y 491.28,Z 691.44,A -85,B 0,C 180,E1 6298.238,E2 6298.238} C_VEL
LIN {X 0,Y 491.215,Z 691.44,A -85,B 0,C 180,E1 6303.538,E2 6303.538} C_VEL
LIN {X 0,Y 491.02,Z 691.44,A -85,B 0,C 180,E1 6309.345,E2 6309.345} C_VEL
LIN {X 0,Y 490.991,Z 691.44,A -85,B 0,C 180,E1 6314.285,E2 6314.285} C_VEL
LIN {X 0,Y 490.877,Z 691.44,A -85,B 0,C 180,E1 6319.835,E2 6319.835} C_VEL
LIN {X 0,Y 490.786,Z 691.44,A -85,B 0,C 180,E1 6325.589,E2 6325.589} C_VEL
LIN {X 0,Y 490.628,Z 691.44,A -85,B 0,C 180,E1 6331.643,E2 6331.643} C_VEL
LIN {X 0,Y 490.598,Z 691.44,A -85,B 0,C 180,E1 6338.114,E2 6338.114} C_VEL
LIN {X 0,Y 490.565,Z 691.44,A -85,B 0,C 180,E1 6344.013,E2 6344.013} C_VEL
LIN {X 0,Y 490.645,Z 691.452,A -85,B 0,C 180,E1 6346.601,E2 6346.601} C_VEL
LIN {X 0,Y 493.198,Z 696.03,A -85,B 0,C 180,E1 6346.993,E2 6346.993} C_VEL
LIN {X 0,Y 494.39,Z 712.797,A -85,B 0,C 180,E1 6347.451,E2 6347.451} C_VEL
LIN {X 0,Y 494.662,Z 713.507,A -85,B 0,C 180,E1 6347.495,E2 6347.495} C_VEL
LIN {X 0,Y 508.939,Z 741.659,A -85,B 0,C 180,E1 6349.494,E2 6349.494} C_VEL
LIN {X 0,Y 506.559,Z 783.383,A -85,B 0,C 180,E1 6350.681,E2 6350.681} C_VEL
LIN {X 0,Y 503.204,Z 824.108,A -85,B 0,C 180,E1 6352.546,E2 6352.546} C_VEL
LIN {X 0,Y 499.288,Z 861.191,A -85,B 0,C 180,E1 6354.958,E2 6354.958} C_VEL
LIN {X 0,Y 495.171,Z 896.573,A -85,B 0,C 180,E1 6358.041,E2 6358.041} C_VEL
LIN {X 0,Y 491.046,Z 930.274,A -85,B 0,C 180,E1 6361.897,E2 6361.897} C_VEL
LIN {X 0,Y 487.801,Z 959.04,A -85,B 0,C 180,E1 6366.203,E2 6366.203} C_VEL
LIN {X 0,Y 485.512,Z 982.848,A -85,B 0,C 180,E1 6370.887,E2 6370.887} C_VEL
LIN {X 0,Y 484.402,Z 1000.808,A -85,B 0,C 180,E1 6375.673,E2 6375.673} C_VEL
LIN {X 0,Y 483.885,Z 1013.234,A -85,B 0,C 180,E1 6380.482,E2 6380.482} C_VEL
LIN {X 0,Y 483.724,Z 1019.905,A -85,B 0,C 180,E1 6384.612,E2 6384.612} C_VEL
LIN {X 0,Y 483.719,Z 1022.657,A -85,B 0,C 180,E1 6388.207,E2 6388.207} C_VEL
LIN {X 0,Y 483.585,Z 1022.657,A -85,B 0,C 180,E1 6391.795,E2 6391.795} C_VEL
LIN {X 0,Y 483.733,Z 1018.703,A -85,B 0,C 180,E1 6396.29,E2 6396.29} C_VEL
LIN {X 0,Y 483.979,Z 1010.435,A -85,B 0,C 180,E1 6400.819,E2 6400.819} C_VEL
LIN {X 0,Y 484.664,Z 995.679,A -85,B 0,C 180,E1 6405.864,E2 6405.864} C_VEL
LIN {X 0,Y 486.254,Z 975.068,A -85,B 0,C 180,E1 6410.796,E2 6410.796} C_VEL
LIN {X 0,Y 488.923,Z 948.93,A -85,B 0,C 180,E1 6415.447,E2 6415.447} C_VEL
LIN {X 0,Y 492.586,Z 917.917,A -85,B 0,C 180,E1 6419.645,E2 6419.645} C_VEL
LIN {X 0,Y 497.012,Z 881.534,A -85,B 0,C 180,E1 6423.375,E2 6423.375} C_VEL
LIN {X 0,Y 501.206,Z 844.474,A -85,B 0,C 180,E1 6426.227,E2 6426.227} C_VEL
LIN {X 0,Y 504.954,Z 805.644,A -85,B 0,C 180,E1 6428.385,E2 6428.385} C_VEL
LIN {X 0,Y 507.721,Z 765.877,A -85,B 0,C 180,E1 6429.896,E2 6429.896} C_VEL
LIN {X 0,Y 508.544,Z 739.549,A -85,B 0,C 180,E1 6430.589,E2 6430.589} C_VEL
LIN {X 0,Y 484.631,Z 696.6,A -85,B 0,C 180,E1 6433.93,E2 6433.93} C_VEL
LIN {X 0,Y 482.742,Z 691.44,A -85,B 0,C 180,E1 6434.285,E2 6434.285} C_VEL
LIN {X 0,Y 482.673,Z 691.44,A -85,B 0,C 180,E1 6441.144,E2 6441.144} C_VEL
LIN {X 0,Y 482.724,Z 691.44,A -85,B 0,C 180,E1 6447.873,E2 6447.873} C_VEL
LIN {X 0,Y 482.844,Z 691.44,A -85,B 0,C 180,E1 6453.959,E2 6453.959} C_VEL
LIN {X 0,Y 483.037,Z 691.44,A -85,B 0,C 180,E1 6460.112,E2 6460.112} C_VEL
LIN {X 0,Y 482.865,Z 691.44,A -85,B 0,C 180,E1 6466.421,E2 6466.421} C_VEL
LIN {X 0,Y 483.289,Z 691.44,A -85,B 0,C 180,E1 6472.798,E2 6472.798} C_VEL
LIN {X 0,Y 483.568,Z 691.44,A -85,B 0,C 180,E1 6478.202,E2 6478.202} C_VEL
LIN {X 0,Y 483.435,Z 691.44,A -85,B 0,C 180,E1 6483.586,E2 6483.586} C_VEL
LIN {X 0,Y 483.235,Z 691.44,A -85,B 0,C 180,E1 6489.007,E2 6489.007} C_VEL
LIN {X 0,Y 483.108,Z 691.44,A -85,B 0,C 180,E1 6494.514,E2 6494.514} C_VEL
LIN {X 0,Y 482.984,Z 691.44,A -85,B 0,C 180,E1 6500.164,E2 6500.164} C_VEL
LIN {X 0,Y 482.845,Z 691.44,A -85,B 0,C 180,E1 6506.032,E2 6506.032} C_VEL
LIN {X 0,Y 482.789,Z 691.44,A -85,B 0,C 180,E1 6512.208,E2 6512.208} C_VEL
LIN {X 0,Y 482.711,Z 691.44,A -85,B 0,C 180,E1 6518.841,E2 6518.841} C_VEL
LIN {X 0,Y 482.631,Z 691.44,A -85,B 0,C 180,E1 6526.167,E2 6526.167} C_VEL
LIN {X 0,Y 485.418,Z 697.419,A -85,B 0,C 180,E1 6526.658,E2 6526.658} C_VEL
LIN {X 0,Y 504.863,Z 734.284,A -85,B 0,C 180,E1 6529.697,E2 6529.697} C_VEL
LIN {X 0,Y 507.541,Z 740.3,A -85,B 0,C 180,E1 6530.171,E2 6530.171} C_VEL
LIN {X 0,Y 504.541,Z 780.066,A -85,B 0,C 180,E1 6531.766,E2 6531.766} C_VEL
LIN {X 0,Y 500.919,Z 816.799,A -85,B 0,C 180,E1 6533.887,E2 6533.887} C_VEL
LIN {X 0,Y 496.641,Z 854.249,A -85,B 0,C 180,E1 6536.821,E2 6536.821} C_VEL
LIN {X 0,Y 492.473,Z 888.266,A -85,B 0,C 180,E1 6540.348,E2 6540.348} C_VEL
LIN {X 0,Y 488.884,Z 919.2,A -85,B 0,C 180,E1 6544.55,E2 6544.55} C_VEL
LIN {X 0,Y 486.228,Z 945.207,A -85,B 0,C 180,E1 6549.188,E2 6549.188} C_VEL
LIN {X 0,Y 484.652,Z 965.829,A -85,B 0,C 180,E1 6554.136,E2 6554.136} C_VEL
LIN {X 0,Y 483.969,Z 980.547,A -85,B 0,C 180,E1 6559.181,E2 6559.181} C_VEL
LIN {X 0,Y 483.747,Z 988.763,A -85,B 0,C 180,E1 6563.71,E2 6563.71} C_VEL
LIN {X 0,Y 483.621,Z 992.673,A -85,B 0,C 180,E1 6568.206,E2 6568.206} C_VEL
LIN {X 0,Y 483.651,Z 992.637,A -85,B 0,C 180,E1 6571.794,E2 6571.794} C_VEL
LIN {X 0,Y 483.71,Z 988.643,A -85,B 0,C 180,E1 6576.289,E2 6576.289} C_VEL
LIN {X 0,Y 483.946,Z 980.323,A -85,B 0,C 180,E1 6580.819,E2 6580.819} C_VEL
LIN {X 0,Y 484.628,Z 965.531,A -85,B 0,C 180,E1 6585.865,E2 6585.865} C_VEL
LIN {X 0,Y 486.088,Z 946.169,A -85,B 0,C 180,E1 6590.52,E2 6590.52} C_VEL
LIN {X 0,Y 488.598,Z 921.601,A -85,B 0,C 180,E1 6594.974,E2 6594.974} C_VEL
LIN {X 0,Y 492.043,Z 892.278,A -85,B 0,C 180,E1 6599.062,E2 6599.062} C_VEL
LIN {X 0,Y 495.95,Z 859.678,A -85,B 0,C 180,E1 6602.581,E2 6602.581} C_VEL
LIN {X 0,Y 500.081,Z 824.609,A -85,B 0,C 180,E1 6605.48,E2 6605.48} C_VEL
LIN {X 0,Y 504.071,Z 785.647,A -85,B 0,C 180,E1 6607.87,E2 6607.87} C_VEL
LIN {X 0,Y 507.274,Z 745.684,A -85,B 0,C 180,E1 6609.56,E2 6609.56} C_VEL
LIN {X 0,Y 506.949,Z 739.357,A -85,B 0,C 180,E1 6609.829,E2 6609.829} C_VEL
LIN {X 0,Y 488.27,Z 702.56,A -85,B 0,C 180,E1 6612.826,E2 6612.826} C_VEL
LIN {X 0,Y 482.846,Z 692.802,A -85,B 0,C 180,E1 6613.636,E2 6613.636} C_VEL
LIN {X 0,Y 482.717,Z 691.44,A -85,B 0,C 180,E1 6613.843,E2 6613.843} C_VEL
LIN {X 0,Y 482.687,Z 691.44,A -85,B 0,C 180,E1 6618.835,E2 6618.835} C_VEL
LIN {X 0,Y 482.605,Z 691.44,A -85,B 0,C 180,E1 6624.656,E2 6624.656} C_VEL
LIN {X 0,Y 482.704,Z 691.44,A -85,B 0,C 180,E1 6629.886,E2 6629.886} C_VEL
LIN {X 0,Y 482.885,Z 691.44,A -85,B 0,C 180,E1 6635.953,E2 6635.953} C_VEL
LIN {X 0,Y 483.039,Z 691.44,A -85,B 0,C 180,E1 6641.74,E2 6641.74} C_VEL
LIN {X 0,Y 483.171,Z 691.44,A -85,B 0,C 180,E1 6647.335,E2 6647.335} C_VEL
LIN {X 0,Y 483.238,Z 691.44,A -85,B 0,C 180,E1 6652.806,E2 6652.806} C_VEL
LIN {X 0,Y 483.395,Z 691.44,A -85,B 0,C 180,E1 6658.21,E2 6658.21} C_VEL
LIN {X 0,Y 483.32,Z 691.44,A -85,B 0,C 180,E1 6663.596,E2 6663.596} C_VEL
LIN {X 0,Y 483.149,Z 691.44,A -85,B 0,C 180,E1 6669.018,E2 6669.018} C_VEL
LIN {X 0,Y 483.072,Z 691.44,A -85,B 0,C 180,E1 6674.524,E2 6674.524} C_VEL
LIN {X 0,Y 482.961,Z 691.44,A -85,B 0,C 180,E1 6680.174,E2 6680.174} C_VEL
LIN {X 0,Y 482.869,Z 691.44,A -85,B 0,C 180,E1 6686.04,E2 6686.04} C_VEL
LIN {X 0,Y 482.683,Z 691.44,A -85,B 0,C 180,E1 6692.226,E2 6692.226} C_VEL
LIN {X 0,Y 482.671,Z 691.44,A -85,B 0,C 180,E1 6698.856,E2 6698.856} C_VEL
LIN {X 0,Y 482.751,Z 691.44,A -85,B 0,C 180,E1 6705.717,E2 6705.717} C_VEL
LIN {X 0,Y 485.274,Z 697.244,A -85,B 0,C 180,E1 6706.156,E2 6706.156} C_VEL
LIN {X 0,Y 494.662,Z 713.507,A -85,B 0,C 180,E1 6707.495,E2 6707.495} C_VEL
LIN {X 0,Y 498.33,Z 734.374,A -85,B 0,C 180,E1 6708.293,E2 6708.293} C_VEL
LIN {X 0,Y 498.87,Z 735.549,A -85,B 0,C 180,E1 6708.374,E2 6708.374} C_VEL
LIN {X 0,Y 502.764,Z 744.769,A -85,B 0,C 180,E1 6708.977,E2 6708.977} C_VEL
LIN {X 0,Y 499.96,Z 788.255,A -85,B 0,C 180,E1 6710.285,E2 6710.285} C_VEL
LIN {X 0,Y 496.013,Z 830.991,A -85,B 0,C 180,E1 6712.375,E2 6712.375} C_VEL
LIN {X 0,Y 491.512,Z 870.501,A -85,B 0,C 180,E1 6715.143,E2 6715.143} C_VEL
LIN {X 0,Y 486.883,Z 907.075,A -85,B 0,C 180,E1 6718.633,E2 6718.633} C_VEL
LIN {X 0,Y 482.614,Z 940.13,A -85,B 0,C 180,E1 6722.809,E2 6722.809} C_VEL
LIN {X 0,Y 479.479,Z 967.388,A -85,B 0,C 180,E1 6727.33,E2 6727.33} C_VEL
LIN {X 0,Y 477.416,Z 990.144,A -85,B 0,C 180,E1 6732.369,E2 6732.369} C_VEL
LIN {X 0,Y 476.31,Z 1005.769,A -85,B 0,C 180,E1 6737.144,E2 6737.144} C_VEL
LIN {X 0,Y 475.888,Z 1015.918,A -85,B 0,C 180,E1 6741.769,E2 6741.769} C_VEL
LIN {X 0,Y 475.705,Z 1021.627,A -85,B 0,C 180,E1 6746.351,E2 6746.351} C_VEL
LIN {X 0,Y 475.73,Z 1023,A -85,B 0,C 180,E1 6750,E2 6750} C_VEL
LIN {X 0,Y 475.704,Z 1021.627,A -85,B 0,C 180,E1 6753.65,E2 6753.65} C_VEL
LIN {X 0,Y 475.901,Z 1015.917,A -85,B 0,C 180,E1 6758.232,E2 6758.232} C_VEL
LIN {X 0,Y 476.233,Z 1005.768,A -85,B 0,C 180,E1 6762.859,E2 6762.859} C_VEL
LIN {X 0,Y 477.406,Z 989.001,A -85,B 0,C 180,E1 6767.938,E2 6767.938} C_VEL
LIN {X 0,Y 479.558,Z 966.327,A -85,B 0,C 180,E1 6772.877,E2 6772.877} C_VEL
LIN {X 0,Y 482.876,Z 937.881,A -85,B 0,C 180,E1 6777.517,E2 6777.517} C_VEL
LIN {X 0,Y 487.142,Z 904.756,A -85,B 0,C 180,E1 6781.617,E2 6781.617} C_VEL
LIN {X 0,Y 491.844,Z 868.049,A -85,B 0,C 180,E1 6785.049,E2 6785.049} C_VEL
LIN {X 0,Y 496.271,Z 829.277,A -85,B 0,C 180,E1 6787.719,E2 6787.719} C_VEL
LIN {X 0,Y 500.139,Z 787.067,A -85,B 0,C 180,E1 6789.754,E2 6789.754} C_VEL
LIN {X 0,Y 502.873,Z 746.591,A -85,B 0,C 180,E1 6790.959,E2 6790.959} C_VEL
LIN {X 0,Y 501.828,Z 741.253,A -85,B 0,C 180,E1 6791.204,E2 6791.204} C_VEL
LIN {X 0,Y 477.356,Z 697.25,A -85,B 0,C 180,E1 6794.756,E2 6794.756} C_VEL
LIN {X 0,Y 474.808,Z 691.44,A -85,B 0,C 180,E1 6795.263,E2 6795.263} C_VEL
LIN {X 0,Y 474.69,Z 691.44,A -85,B 0,C 180,E1 6800.364,E2 6800.364} C_VEL
LIN {X 0,Y 474.699,Z 691.44,A -85,B 0,C 180,E1 6806.026,E2 6806.026} C_VEL
LIN {X 0,Y 474.783,Z 691.44,A -85,B 0,C 180,E1 6811.422,E2 6811.422} C_VEL
LIN {X 0,Y 475.027,Z 691.44,A -85,B 0,C 180,E1 6817.569,E2 6817.569} C_VEL
LIN {X 0,Y 475.043,Z 691.44,A -85,B 0,C 180,E1 6823.328,E2 6823.328} C_VEL
LIN {X 0,Y 475.125,Z 691.44,A -85,B 0,C 180,E1 6828.974,E2 6828.974} C_VEL
LIN {X 0,Y 475.437,Z 691.44,A -85,B 0,C 180,E1 6834.514,E2 6834.514} C_VEL
LIN {X 0,Y 475.553,Z 691.44,A -85,B 0,C 180,E1 6839.996,E2 6839.996} C_VEL
LIN {X 0,Y 475.407,Z 691.44,A -85,B 0,C 180,E1 6845.477,E2 6845.477} C_VEL
LIN {X 0,Y 475.24,Z 691.44,A -85,B 0,C 180,E1 6851.014,E2 6851.014} C_VEL
LIN {X 0,Y 475.098,Z 691.44,A -85,B 0,C 180,E1 6857.046,E2 6857.046} C_VEL
LIN {X 0,Y 475.006,Z 691.44,A -85,B 0,C 180,E1 6862.481,E2 6862.481} C_VEL
LIN {X 0,Y 474.83,Z 691.44,A -85,B 0,C 180,E1 6868.565,E2 6868.565} C_VEL
LIN {X 0,Y 474.824,Z 691.44,A -85,B 0,C 180,E1 6875.017,E2 6875.017} C_VEL
LIN {X 0,Y 474.67,Z 691.44,A -85,B 0,C 180,E1 6880.044,E2 6880.044} C_VEL
LIN {X 0,Y 474.606,Z 691.44,A -85,B 0,C 180,E1 6885.265,E2 6885.265} C_VEL
LIN {X 0,Y 477.177,Z 697.207,A -85,B 0,C 180,E1 6885.705,E2 6885.705} C_VEL
LIN {X 0,Y 496.058,Z 731.595,A -85,B 0,C 180,E1 6888.715,E2 6888.715} C_VEL
LIN {X 0,Y 501.19,Z 744.61,A -85,B 0,C 180,E1 6889.713,E2 6889.713} C_VEL
LIN {X 0,Y 497.556,Z 788.126,A -85,B 0,C 180,E1 6891.588,E2 6891.588} C_VEL
LIN {X 0,Y 492.932,Z 828.697,A -85,B 0,C 180,E1 6894.172,E2 6894.172} C_VEL
LIN {X 0,Y 488.355,Z 865.594,A -85,B 0,C 180,E1 6897.383,E2 6897.383} C_VEL
LIN {X 0,Y 483.888,Z 899.628,A -85,B 0,C 180,E1 6901.305,E2 6901.305} C_VEL
LIN {X 0,Y 480.365,Z 929.282,A -85,B 0,C 180,E1 6905.81,E2 6905.81} C_VEL
LIN {X 0,Y 477.925,Z 953.027,A -85,B 0,C 180,E1 6910.57,E2 6910.57} C_VEL
LIN {X 0,Y 476.594,Z 971.315,A -85,B 0,C 180,E1 6915.551,E2 6915.551} C_VEL
LIN {X 0,Y 475.909,Z 984.418,A -85,B 0,C 180,E1 6920.847,E2 6920.847} C_VEL
LIN {X 0,Y 475.764,Z 989.955,A -85,B 0,C 180,E1 6924.521,E2 6924.521} C_VEL
LIN {X 0,Y 475.719,Z 992.672,A -85,B 0,C 180,E1 6928.176,E2 6928.176} C_VEL
LIN {X 0,Y 475.745,Z 992.637,A -85,B 0,C 180,E1 6931.823,E2 6931.823} C_VEL
LIN {X 0,Y 475.8,Z 988.644,A -85,B 0,C 180,E1 6936.394,E2 6936.394} C_VEL
LIN {X 0,Y 476.07,Z 980.325,A -85,B 0,C 180,E1 6941,E2 6941} C_VEL
LIN {X 0,Y 476.867,Z 965.534,A -85,B 0,C 180,E1 6946.13,E2 6946.13} C_VEL
LIN {X 0,Y 478.657,Z 945.058,A -85,B 0,C 180,E1 6951.1,E2 6951.1} C_VEL
LIN {X 0,Y 481.58,Z 918.669,A -85,B 0,C 180,E1 6955.863,E2 6955.863} C_VEL
LIN {X 0,Y 485.629,Z 886.426,A -85,B 0,C 180,E1 6960.254,E2 6960.254} C_VEL
LIN {X 0,Y 490.197,Z 851.188,A -85,B 0,C 180,E1 6963.889,E2 6963.889} C_VEL
LIN {X 0,Y 494.988,Z 812.17,A -85,B 0,C 180,E1 6966.893,E2 6966.893} C_VEL
LIN {X 0,Y 499.128,Z 772.129,A -85,B 0,C 180,E1 6969.105,E2 6969.105} C_VEL
LIN {X 0,Y 500.856,Z 742.727,A -85,B 0,C 180,E1 6970.302,E2 6970.302} C_VEL
LIN {X 0,Y 482.962,Z 707.105,A -85,B 0,C 180,E1 6973.312,E2 6973.312} C_VEL
LIN {X 0,Y 474.811,Z 692.473,A -85,B 0,C 180,E1 6974.585,E2 6974.585} C_VEL
LIN {X 0,Y 474.718,Z 691.44,A -85,B 0,C 180,E1 6974.623,E2 6974.623} C_VEL
LIN {X 0,Y 474.672,Z 691.44,A -85,B 0,C 180,E1 6980.373,E2 6980.373} C_VEL
LIN {X 0,Y 474.692,Z 691.44,A -85,B 0,C 180,E1 6987.175,E2 6987.175} C_VEL
LIN {X 0,Y 474.878,Z 691.44,A -85,B 0,C 180,E1 6993.498,E2 6993.498} C_VEL
LIN {X 0,Y 475.057,Z 691.44,A -85,B 0,C 180,E1 6999.484,E2 6999.484} C_VEL
LIN {X 0,Y 475.262,Z 691.44,A -85,B 0,C 180,E1 7005.241,E2 7005.241} C_VEL
LIN {X 0,Y 475.341,Z 691.44,A -85,B 0,C 180,E1 7011.194,E2 7011.194} C_VEL
LIN {X 0,Y 475.579,Z 691.44,A -85,B 0,C 180,E1 7016.354,E2 7016.354} C_VEL
LIN {X 0,Y 475.678,Z 691.44,A -85,B 0,C 180,E1 7021.828,E2 7021.828} C_VEL
LIN {X 0,Y 475.366,Z 691.44,A -85,B 0,C 180,E1 7027.323,E2 7027.323} C_VEL
LIN {X 0,Y 475.18,Z 691.44,A -85,B 0,C 180,E1 7032.891,E2 7032.891} C_VEL
LIN {X 0,Y 475.05,Z 691.44,A -85,B 0,C 180,E1 7038.588,E2 7038.588} C_VEL
LIN {X 0,Y 474.985,Z 691.44,A -85,B 0,C 180,E1 7044.482,E2 7044.482} C_VEL
LIN {X 0,Y 474.753,Z 691.44,A -85,B 0,C 180,E1 7050.682,E2 7050.682} C_VEL
LIN {X 0,Y 474.735,Z 691.44,A -85,B 0,C 180,E1 7057.298,E2 7057.298} C_VEL
LIN {X 0,Y 474.68,Z 691.44,A -85,B 0,C 180,E1 7062.809,E2 7062.809} C_VEL
LIN {X 0,Y 474.844,Z 691.44,A -85,B 0,C 180,E1 7064.793,E2 7064.793} C_VEL
LIN {X 0,Y 477.366,Z 697.25,A -85,B 0,C 180,E1 7065.246,E2 7065.246} C_VEL
LIN {X 0,Y 498.87,Z 735.549,A -85,B 0,C 180,E1 7068.374,E2 7068.374} C_VEL
LIN {X 0,Y 499.72,Z 742.24,A -85,B 0,C 180,E1 7068.608,E2 7068.608} C_VEL
LIN {X 0,Y 495.97,Z 758.872,A -85,B 0,C 180,E1 7068.725,E2 7068.725} C_VEL
LIN {X 0,Y 492.615,Z 802.457,A -85,B 0,C 180,E1 7070.318,E2 7070.318} C_VEL
LIN {X 0,Y 488.167,Z 843.794,A -85,B 0,C 180,E1 7072.625,E2 7072.625} C_VEL
LIN {X 0,Y 483.211,Z 882.777,A -85,B 0,C 180,E1 7075.667,E2 7075.667} C_VEL
LIN {X 0,Y 478.306,Z 918.301,A -85,B 0,C 180,E1 7079.428,E2 7079.428} C_VEL
LIN {X 0,Y 474.188,Z 948.937,A -85,B 0,C 180,E1 7083.703,E2 7083.703} C_VEL
LIN {X 0,Y 471.034,Z 975.354,A -85,B 0,C 180,E1 7088.562,E2 7088.562} C_VEL
LIN {X 0,Y 469.12,Z 995.684,A -85,B 0,C 180,E1 7093.597,E2 7093.597} C_VEL
LIN {X 0,Y 468.147,Z 1010.436,A -85,B 0,C 180,E1 7098.811,E2 7098.811} C_VEL
LIN {X 0,Y 467.92,Z 1018.703,A -85,B 0,C 180,E1 7103.498,E2 7103.498} C_VEL
LIN {X 0,Y 467.92,Z 1022.657,A -85,B 0,C 180,E1 7108.146,E2 7108.146} C_VEL
LIN {X 0,Y 467.783,Z 1022.657,A -85,B 0,C 180,E1 7111.855,E2 7111.855} C_VEL
LIN {X 0,Y 467.929,Z 1018.703,A -85,B 0,C 180,E1 7116.503,E2 7116.503} C_VEL
LIN {X 0,Y 468.218,Z 1010.434,A -85,B 0,C 180,E1 7121.188,E2 7121.188} C_VEL
LIN {X 0,Y 469.089,Z 995.681,A -85,B 0,C 180,E1 7126.405,E2 7126.405} C_VEL
LIN {X 0,Y 471.098,Z 974.57,A -85,B 0,C 180,E1 7131.609,E2 7131.609} C_VEL
LIN {X 0,Y 474.165,Z 948.933,A -85,B 0,C 180,E1 7136.299,E2 7136.299} C_VEL
LIN {X 0,Y 478.484,Z 917.223,A -85,B 0,C 180,E1 7140.7,E2 7140.7} C_VEL
LIN {X 0,Y 483.426,Z 881.725,A -85,B 0,C 180,E1 7144.42,E2 7144.42} C_VEL
LIN {X 0,Y 488.263,Z 843.522,A -85,B 0,C 180,E1 7147.388,E2 7147.388} C_VEL
LIN {X 0,Y 492.722,Z 801.781,A -85,B 0,C 180,E1 7149.71,E2 7149.71} C_VEL
LIN {X 0,Y 495.859,Z 762.564,A -85,B 0,C 180,E1 7151.151,E2 7151.151} C_VEL
LIN {X 0,Y 496.326,Z 745.479,A -85,B 0,C 180,E1 7151.642,E2 7151.642} C_VEL
LIN {X 0,Y 472.897,Z 702.939,A -85,B 0,C 180,E1 7155.17,E2 7155.17} C_VEL
LIN {X 0,Y 466.924,Z 692.708,A -85,B 0,C 180,E1 7156.126,E2 7156.126} C_VEL
LIN {X 0,Y 466.781,Z 691.44,A -85,B 0,C 180,E1 7156.289,E2 7156.289} C_VEL
LIN {X 0,Y 466.738,Z 691.44,A -85,B 0,C 180,E1 7161.95,E2 7161.95} C_VEL
LIN {X 0,Y 466.785,Z 691.44,A -85,B 0,C 180,E1 7168.736,E2 7168.736} C_VEL
LIN {X 0,Y 467.007,Z 691.44,A -85,B 0,C 180,E1 7175.202,E2 7175.202} C_VEL
LIN {X 0,Y 467.15,Z 691.44,A -85,B 0,C 180,E1 7181.086,E2 7181.086} C_VEL
LIN {X 0,Y 467.082,Z 691.44,A -85,B 0,C 180,E1 7186.882,E2 7186.882} C_VEL
LIN {X 0,Y 467.436,Z 691.44,A -85,B 0,C 180,E1 7192.552,E2 7192.552} C_VEL
LIN {X 0,Y 467.759,Z 691.44,A -85,B 0,C 180,E1 7198.141,E2 7198.141} C_VEL
LIN {X 0,Y 467.609,Z 691.44,A -85,B 0,C 180,E1 7203.708,E2 7203.708} C_VEL
LIN {X 0,Y 467.407,Z 691.44,A -85,B 0,C 180,E1 7209.315,E2 7209.315} C_VEL
LIN {X 0,Y 467.235,Z 691.44,A -85,B 0,C 180,E1 7215.018,E2 7215.018} C_VEL
LIN {X 0,Y 467.105,Z 691.44,A -85,B 0,C 180,E1 7220.881,E2 7220.881} C_VEL
LIN {X 0,Y 466.935,Z 691.44,A -85,B 0,C 180,E1 7226.989,E2 7226.989} C_VEL
LIN {X 0,Y 466.876,Z 691.44,A -85,B 0,C 180,E1 7233.446,E2 7233.446} C_VEL
LIN {X 0,Y 466.72,Z 691.44,A -85,B 0,C 180,E1 7240.44,E2 7240.44} C_VEL
LIN {X 0,Y 466.681,Z 691.916,A -85,B 0,C 180,E1 7244.308,E2 7244.308} C_VEL
LIN {X 0,Y 469.371,Z 697.367,A -85,B 0,C 180,E1 7244.763,E2 7244.763} C_VEL
LIN {X 0,Y 488.899,Z 732.477,A -85,B 0,C 180,E1 7247.995,E2 7247.995} C_VEL
LIN {X 0,Y 495.039,Z 746.443,A -85,B 0,C 180,E1 7249.175,E2 7249.175} C_VEL
LIN {X 0,Y 491.219,Z 789.285,A -85,B 0,C 180,E1 7251.058,E2 7251.058} C_VEL
LIN {X 0,Y 486.415,Z 829.212,A -85,B 0,C 180,E1 7253.636,E2 7253.636} C_VEL
LIN {X 0,Y 481.329,Z 866.608,A -85,B 0,C 180,E1 7256.966,E2 7256.966} C_VEL
LIN {X 0,Y 476.684,Z 899.622,A -85,B 0,C 180,E1 7260.83,E2 7260.83} C_VEL
LIN {X 0,Y 472.841,Z 929.279,A -85,B 0,C 180,E1 7265.4,E2 7265.4} C_VEL
LIN {X 0,Y 470.209,Z 953.026,A -85,B 0,C 180,E1 7270.238,E2 7270.238} C_VEL
LIN {X 0,Y 468.806,Z 970.439,A -85,B 0,C 180,E1 7275.026,E2 7275.026} C_VEL
LIN {X 0,Y 468.118,Z 983.383,A -85,B 0,C 180,E1 7280.186,E2 7280.186} C_VEL
LIN {X 0,Y 467.868,Z 989.954,A -85,B 0,C 180,E1 7284.428,E2 7284.428} C_VEL
LIN {X 0,Y 467.832,Z 992.672,A -85,B 0,C 180,E1 7288.145,E2 7288.145} C_VEL
LIN {X 0,Y 467.851,Z 992.638,A -85,B 0,C 180,E1 7291.854,E2 7291.854} C_VEL
LIN {X 0,Y 467.891,Z 988.645,A -85,B 0,C 180,E1 7296.503,E2 7296.503} C_VEL
LIN {X 0,Y 468.183,Z 980.326,A -85,B 0,C 180,E1 7301.188,E2 7301.188} C_VEL
LIN {X 0,Y 469.093,Z 965.537,A -85,B 0,C 180,E1 7306.404,E2 7306.404} C_VEL
LIN {X 0,Y 471.041,Z 945.08,A -85,B 0,C 180,E1 7311.454,E2 7311.454} C_VEL
LIN {X 0,Y 474.205,Z 918.675,A -85,B 0,C 180,E1 7316.296,E2 7316.296} C_VEL
LIN {X 0,Y 478.507,Z 886.808,A -85,B 0,C 180,E1 7320.706,E2 7320.706} C_VEL
LIN {X 0,Y 483.452,Z 851.293,A -85,B 0,C 180,E1 7324.424,E2 7324.424} C_VEL
LIN {X 0,Y 488.494,Z 813.578,A -85,B 0,C 180,E1 7327.386,E2 7327.386} C_VEL
LIN {X 0,Y 492.925,Z 773.104,A -85,B 0,C 180,E1 7329.659,E2 7329.659} C_VEL
LIN {X 0,Y 494.651,Z 745.752,A -85,B 0,C 180,E1 7330.805,E2 7330.805} C_VEL
LIN {X 0,Y 477.667,Z 711.501,A -85,B 0,C 180,E1 7333.813,E2 7333.813} C_VEL
LIN {X 0,Y 466.926,Z 692.939,A -85,B 0,C 180,E1 7335.547,E2 7335.547} C_VEL
LIN {X 0,Y 466.793,Z 691.44,A -85,B 0,C 180,E1 7335.71,E2 7335.71} C_VEL
LIN {X 0,Y 466.709,Z 691.44,A -85,B 0,C 180,E1 7341.959,E2 7341.959} C_VEL
LIN {X 0,Y 466.774,Z 691.44,A -85,B 0,C 180,E1 7348.745,E2 7348.745} C_VEL
LIN {X 0,Y 467.042,Z 691.44,A -85,B 0,C 180,E1 7355.191,E2 7355.191} C_VEL
LIN {X 0,Y 467.162,Z 691.44,A -85,B 0,C 180,E1 7361.096,E2 7361.096} C_VEL
LIN {X 0,Y 467.337,Z 691.44,A -85,B 0,C 180,E1 7366.898,E2 7366.898} C_VEL
LIN {X 0,Y 467.416,Z 691.44,A -85,B 0,C 180,E1 7372.561,E2 7372.561} C_VEL
LIN {X 0,Y 467.623,Z 691.44,A -85,B 0,C 180,E1 7378.149,E2 7378.149} C_VEL
LIN {X 0,Y 467.507,Z 691.44,A -85,B 0,C 180,E1 7383.718,E2 7383.718} C_VEL
LIN {X 0,Y 467.311,Z 691.44,A -85,B 0,C 180,E1 7389.326,E2 7389.326} C_VEL
LIN {X 0,Y 467.205,Z 691.44,A -85,B 0,C 180,E1 7395.029,E2 7395.029} C_VEL
LIN {X 0,Y 467.096,Z 691.44,A -85,B 0,C 180,E1 7400.891,E2 7400.891} C_VEL
LIN {X 0,Y 466.943,Z 691.44,A -85,B 0,C 180,E1 7406.999,E2 7406.999} C_VEL
LIN {X 0,Y 466.769,Z 691.44,A -85,B 0,C 180,E1 7413.466,E2 7413.466} C_VEL
LIN {X 0,Y 466.745,Z 691.44,A -85,B 0,C 180,E1 7420.449,E2 7420.449} C_VEL
LIN {X 0,Y 466.83,Z 691.722,A -85,B 0,C 180,E1 7423.842,E2 7423.842} C_VEL
LIN {X 0,Y 469.296,Z 697.146,A -85,B 0,C 180,E1 7424.268,E2 7424.268} C_VEL
LIN {X 0,Y 492.761,Z 738.397,A -85,B 0,C 180,E1 7427.812,E2 7427.812} C_VEL
LIN {X 0,Y 496.615,Z 747.238,A -85,B 0,C 180,E1 7428.439,E2 7428.439} C_VEL
LIN {X 0,Y 495.97,Z 758.872,A -85,B 0,C 180,E1 7428.725,E2 7428.725} C_VEL
LIN {X 0,Y 491.588,Z 775.824,A -85,B 0,C 180,E1 7428.936,E2 7428.936} C_VEL
LIN {X 0,Y 487.499,Z 790.474,A -85,B 0,C 180,E1 7429.204,E2 7429.204} C_VEL
LIN {X 0,Y 487.245,Z 792.482,A -85,B 0,C 180,E1 7429.284,E2 7429.284} C_VEL
LIN {X 0,Y 482.874,Z 833.345,A -85,B 0,C 180,E1 7431.385,E2 7431.385} C_VEL
LIN {X 0,Y 477.974,Z 871.453,A -85,B 0,C 180,E1 7434.147,E2 7434.147} C_VEL
LIN {X 0,Y 472.706,Z 908.465,A -85,B 0,C 180,E1 7437.76,E2 7437.76} C_VEL
LIN {X 0,Y 468.119,Z 939.368,A -85,B 0,C 180,E1 7441.769,E2 7441.769} C_VEL
LIN {X 0,Y 464.406,Z 966.542,A -85,B 0,C 180,E1 7446.374,E2 7446.374} C_VEL
LIN {X 0,Y 461.959,Z 989.126,A -85,B 0,C 180,E1 7451.472,E2 7451.472} C_VEL
LIN {X 0,Y 460.623,Z 1005.768,A -85,B 0,C 180,E1 7456.698,E2 7456.698} C_VEL
LIN {X 0,Y 460.118,Z 1016.106,A -85,B 0,C 180,E1 7461.599,E2 7461.599} C_VEL
LIN {X 0,Y 459.914,Z 1021.627,A -85,B 0,C 180,E1 7466.225,E2 7466.225} C_VEL
LIN {X 0,Y 459.947,Z 1023,A -85,B 0,C 180,E1 7470,E2 7470} C_VEL
LIN {X 0,Y 459.909,Z 1021.627,A -85,B 0,C 180,E1 7473.776,E2 7473.776} C_VEL
LIN {X 0,Y 460.128,Z 1016.101,A -85,B 0,C 180,E1 7478.404,E2 7478.404} C_VEL
LIN {X 0,Y 460.547,Z 1005.767,A -85,B 0,C 180,E1 7483.305,E2 7483.305} C_VEL
LIN {X 0,Y 461.929,Z 989.24,A -85,B 0,C 180,E1 7488.497,E2 7488.497} C_VEL
LIN {X 0,Y 464.425,Z 966.471,A -85,B 0,C 180,E1 7493.639,E2 7493.639} C_VEL
LIN {X 0,Y 468.393,Z 937.658,A -85,B 0,C 180,E1 7498.477,E2 7498.477} C_VEL
LIN {X 0,Y 473.18,Z 905.469,A -85,B 0,C 180,E1 7502.575,E2 7502.575} C_VEL
LIN {X 0,Y 478.49,Z 867.73,A -85,B 0,C 180,E1 7506.162,E2 7506.162} C_VEL
LIN {X 0,Y 483.662,Z 827.357,A -85,B 0,C 180,E1 7508.971,E2 7508.971} C_VEL
LIN {X 0,Y 487.976,Z 785.35,A -85,B 0,C 180,E1 7511.002,E2 7511.002} C_VEL
LIN {X 0,Y 490.274,Z 748.593,A -85,B 0,C 180,E1 7512.171,E2 7512.171} C_VEL
LIN {X 0,Y 468.31,Z 708.318,A -85,B 0,C 180,E1 7515.617,E2 7515.617} C_VEL
LIN {X 0,Y 459.036,Z 692.87,A -85,B 0,C 180,E1 7517.148,E2 7517.148} C_VEL
LIN {X 0,Y 458.874,Z 691.44,A -85,B 0,C 180,E1 7517.365,E2 7517.365} C_VEL
LIN {X 0,Y 458.796,Z 691.44,A -85,B 0,C 180,E1 7523.557,E2 7523.557} C_VEL
LIN {X 0,Y 458.865,Z 691.44,A -85,B 0,C 180,E1 7530.333,E2 7530.333} C_VEL
LIN {X 0,Y 459.1,Z 691.44,A -85,B 0,C 180,E1 7536.686,E2 7536.686} C_VEL
LIN {X 0,Y 459.231,Z 691.44,A -85,B 0,C 180,E1 7542.967,E2 7542.967} C_VEL
LIN {X 0,Y 459.254,Z 691.44,A -85,B 0,C 180,E1 7548.588,E2 7548.588} C_VEL
LIN {X 0,Y 459.603,Z 691.44,A -85,B 0,C 180,E1 7554.324,E2 7554.324} C_VEL
LIN {X 0,Y 459.771,Z 691.44,A -85,B 0,C 180,E1 7559.995,E2 7559.995} C_VEL
LIN {X 0,Y 459.572,Z 691.44,A -85,B 0,C 180,E1 7565.667,E2 7565.667} C_VEL
LIN {X 0,Y 459.383,Z 691.44,A -85,B 0,C 180,E1 7571.399,E2 7571.399} C_VEL
LIN {X 0,Y 459.286,Z 691.44,A -85,B 0,C 180,E1 7577.252,E2 7577.252} C_VEL
LIN {X 0,Y 459.11,Z 691.44,A -85,B 0,C 180,E1 7583.304,E2 7583.304} C_VEL
LIN {X 0,Y 458.925,Z 691.44,A -85,B 0,C 180,E1 7589.652,E2 7589.652} C_VEL
LIN {X 0,Y 458.868,Z 691.44,A -85,B 0,C 180,E1 7596.425,E2 7596.425} C_VEL
LIN {X 0,Y 458.785,Z 691.44,A -85,B 0,C 180,E1 7603.233,E2 7603.233} C_VEL
LIN {X 0,Y 461.264,Z 697.23,A -85,B 0,C 180,E1 7603.727,E2 7603.727} C_VEL
LIN {X 0,Y 481.012,Z 731.969,A -85,B 0,C 180,E1 7607.109,E2 7607.109} C_VEL
LIN {X 0,Y 488.797,Z 749.441,A -85,B 0,C 180,E1 7608.663,E2 7608.663} C_VEL
LIN {X 0,Y 484.955,Z 790.348,A -85,B 0,C 180,E1 7610.51,E2 7610.51} C_VEL
LIN {X 0,Y 479.965,Z 829.457,A -85,B 0,C 180,E1 7613.063,E2 7613.063} C_VEL
LIN {X 0,Y 474.746,Z 865.613,A -85,B 0,C 180,E1 7616.307,E2 7616.307} C_VEL
LIN {X 0,Y 469.562,Z 899.506,A -85,B 0,C 180,E1 7620.327,E2 7620.327} C_VEL
LIN {X 0,Y 465.366,Z 929.275,A -85,B 0,C 180,E1 7624.978,E2 7624.978} C_VEL
LIN {X 0,Y 462.462,Z 953.023,A -85,B 0,C 180,E1 7629.893,E2 7629.893} C_VEL
LIN {X 0,Y 460.994,Z 970.436,A -85,B 0,C 180,E1 7634.766,E2 7634.766} C_VEL
LIN {X 0,Y 460.267,Z 982.495,A -85,B 0,C 180,E1 7639.576,E2 7639.576} C_VEL
LIN {X 0,Y 459.971,Z 989.954,A -85,B 0,C 180,E1 7644.332,E2 7644.332} C_VEL
LIN {X 0,Y 459.929,Z 992.672,A -85,B 0,C 180,E1 7648.113,E2 7648.113} C_VEL
LIN {X 0,Y 459.944,Z 992.638,A -85,B 0,C 180,E1 7651.886,E2 7651.886} C_VEL
LIN {X 0,Y 459.989,Z 988.646,A -85,B 0,C 180,E1 7656.615,E2 7656.615} C_VEL
LIN {X 0,Y 460.321,Z 980.328,A -85,B 0,C 180,E1 7661.382,E2 7661.382} C_VEL
LIN {X 0,Y 461.338,Z 965.54,A -85,B 0,C 180,E1 7666.688,E2 7666.688} C_VEL
LIN {X 0,Y 463.489,Z 944.546,A -85,B 0,C 180,E1 7671.943,E2 7671.943} C_VEL
LIN {X 0,Y 466.825,Z 918.68,A -85,B 0,C 180,E1 7676.744,E2 7676.744} C_VEL
LIN {X 0,Y 471.429,Z 887.233,A -85,B 0,C 180,E1 7681.164,E2 7681.164} C_VEL
LIN {X 0,Y 476.851,Z 850.847,A -85,B 0,C 180,E1 7685.047,E2 7685.047} C_VEL
LIN {X 0,Y 482.167,Z 813.458,A -85,B 0,C 180,E1 7687.996,E2 7687.996} C_VEL
LIN {X 0,Y 486.933,Z 772.026,A -85,B 0,C 180,E1 7690.32,E2 7690.32} C_VEL
LIN {X 0,Y 488.475,Z 748.803,A -85,B 0,C 180,E1 7691.31,E2 7691.31} C_VEL
LIN {X 0,Y 471.176,Z 713.426,A -85,B 0,C 180,E1 7694.537,E2 7694.537} C_VEL
LIN {X 0,Y 459.044,Z 693.142,A -85,B 0,C 180,E1 7696.565,E2 7696.565} C_VEL
LIN {X 0,Y 458.857,Z 691.44,A -85,B 0,C 180,E1 7696.802,E2 7696.802} C_VEL
LIN {X 0,Y 458.764,Z 691.44,A -85,B 0,C 180,E1 7703.566,E2 7703.566} C_VEL
LIN {X 0,Y 458.856,Z 691.44,A -85,B 0,C 180,E1 7710.343,E2 7710.343} C_VEL
LIN {X 0,Y 459.115,Z 691.44,A -85,B 0,C 180,E1 7716.696,E2 7716.696} C_VEL
LIN {X 0,Y 459.342,Z 691.44,A -85,B 0,C 180,E1 7722.919,E2 7722.919} C_VEL
LIN {X 0,Y 459.439,Z 691.44,A -85,B 0,C 180,E1 7728.602,E2 7728.602} C_VEL
LIN {X 0,Y 459.577,Z 691.44,A -85,B 0,C 180,E1 7734.333,E2 7734.333} C_VEL
LIN {X 0,Y 459.819,Z 691.44,A -85,B 0,C 180,E1 7740.005,E2 7740.005} C_VEL
LIN {X 0,Y 459.609,Z 691.44,A -85,B 0,C 180,E1 7745.676,E2 7745.676} C_VEL
LIN {X 0,Y 459.36,Z 691.44,A -85,B 0,C 180,E1 7751.409,E2 7751.409} C_VEL
LIN {X 0,Y 459.236,Z 691.44,A -85,B 0,C 180,E1 7757.263,E2 7757.263} C_VEL
LIN {X 0,Y 459.123,Z 691.44,A -85,B 0,C 180,E1 7763.313,E2 7763.313} C_VEL
LIN {X 0,Y 458.865,Z 691.44,A -85,B 0,C 180,E1 7769.667,E2 7769.667} C_VEL
LIN {X 0,Y 458.79,Z 691.44,A -85,B 0,C 180,E1 7776.443,E2 7776.443} C_VEL
LIN {X 0,Y 458.927,Z 691.9,A -85,B 0,C 180,E1 7782.819,E2 7782.819} C_VEL
LIN {X 0,Y 461.642,Z 697.435,A -85,B 0,C 180,E1 7783.301,E2 7783.301} C_VEL
LIN {X 0,Y 483.783,Z 735.871,A -85,B 0,C 180,E1 7786.792,E2 7786.792} C_VEL
LIN {X 0,Y 490.544,Z 750.421,A -85,B 0,C 180,E1 7787.912,E2 7787.912} C_VEL
LIN {X 0,Y 487.418,Z 791.035,A -85,B 0,C 180,E1 7789.226,E2 7789.226} C_VEL
LIN {X 0,Y 487.245,Z 792.482,A -85,B 0,C 180,E1 7789.284,E2 7789.284} C_VEL
LIN {X 0,Y 482.539,Z 809.119,A -85,B 0,C 180,E1 7789.748,E2 7789.748} C_VEL
LIN {X 0,Y 477.632,Z 825.084,A -85,B 0,C 180,E1 7790.307,E2 7790.307} C_VEL
LIN {X 0,Y 472.506,Z 863.485,A -85,B 0,C 180,E1 7792.942,E2 7792.942} C_VEL
LIN {X 0,Y 467.266,Z 898.591,A -85,B 0,C 180,E1 7796.178,E2 7796.178} C_VEL
LIN {X 0,Y 462.234,Z 930.794,A -85,B 0,C 180,E1 7800.054,E2 7800.054} C_VEL
LIN {X 0,Y 458.005,Z 959.044,A -85,B 0,C 180,E1 7804.548,E2 7804.548} C_VEL
LIN {X 0,Y 454.786,Z 982.904,A -85,B 0,C 180,E1 7809.552,E2 7809.552} C_VEL
LIN {X 0,Y 453.072,Z 1001.403,A -85,B 0,C 180,E1 7814.862,E2 7814.862} C_VEL
LIN {X 0,Y 452.292,Z 1014.331,A -85,B 0,C 180,E1 7820.365,E2 7820.365} C_VEL
LIN {X 0,Y 452.117,Z 1019.905,A -85,B 0,C 180,E1 7824.234,E2 7824.234} C_VEL
LIN {X 0,Y 452.105,Z 1022.657,A -85,B 0,C 180,E1 7828.081,E2 7828.081} C_VEL
LIN {X 0,Y 451.989,Z 1022.657,A -85,B 0,C 180,E1 7831.92,E2 7831.92} C_VEL
LIN {X 0,Y 452.141,Z 1018.703,A -85,B 0,C 180,E1 7836.731,E2 7836.731} C_VEL
LIN {X 0,Y 452.456,Z 1010.434,A -85,B 0,C 180,E1 7841.583,E2 7841.583} C_VEL
LIN {X 0,Y 453.543,Z 995.683,A -85,B 0,C 180,E1 7846.984,E2 7846.984} C_VEL
LIN {X 0,Y 455.941,Z 974.175,A -85,B 0,C 180,E1 7852.451,E2 7852.451} C_VEL
LIN {X 0,Y 459.662,Z 947.365,A -85,B 0,C 180,E1 7857.462,E2 7857.462} C_VEL
LIN {X 0,Y 464.366,Z 917.279,A -85,B 0,C 180,E1 7861.71,E2 7861.71} C_VEL
LIN {X 0,Y 470.04,Z 880.52,A -85,B 0,C 180,E1 7865.605,E2 7865.605} C_VEL
LIN {X 0,Y 475.569,Z 841.555,A -85,B 0,C 180,E1 7868.67,E2 7868.67} C_VEL
LIN {X 0,Y 480.506,Z 800.852,A -85,B 0,C 180,E1 7870.949,E2 7870.949} C_VEL
LIN {X 0,Y 483.957,Z 762.501,A -85,B 0,C 180,E1 7872.374,E2 7872.374} C_VEL
LIN {X 0,Y 484.175,Z 751.541,A -85,B 0,C 180,E1 7872.727,E2 7872.727} C_VEL
LIN {X 0,Y 463.632,Z 713.561,A -85,B 0,C 180,E1 7876.091,E2 7876.091} C_VEL
LIN {X 0,Y 451.027,Z 692.608,A -85,B 0,C 180,E1 7878.252,E2 7878.252} C_VEL
LIN {X 0,Y 450.945,Z 691.44,A -85,B 0,C 180,E1 7878.384,E2 7878.384} C_VEL
LIN {X 0,Y 450.87,Z 691.44,A -85,B 0,C 180,E1 7885.188,E2 7885.188} C_VEL
LIN {X 0,Y 450.991,Z 691.44,A -85,B 0,C 180,E1 7891.964,E2 7891.964} C_VEL
LIN {X 0,Y 451.226,Z 691.44,A -85,B 0,C 180,E1 7898.338,E2 7898.338} C_VEL
LIN {X 0,Y 451.236,Z 691.44,A -85,B 0,C 180,E1 7904.426,E2 7904.426} C_VEL
LIN {X 0,Y 451.432,Z 691.44,A -85,B 0,C 180,E1 7910.343,E2 7910.343} C_VEL
LIN {X 0,Y 451.693,Z 691.44,A -85,B 0,C 180,E1 7916.152,E2 7916.152} C_VEL
LIN {X 0,Y 451.799,Z 691.44,A -85,B 0,C 180,E1 7921.916,E2 7921.916} C_VEL
LIN {X 0,Y 451.608,Z 691.44,A -85,B 0,C 180,E1 7927.701,E2 7927.701} C_VEL
LIN {X 0,Y 451.424,Z 691.44,A -85,B 0,C 180,E1 7933.572,E2 7933.572} C_VEL
LIN {X 0,Y 451.233,Z 691.44,A -85,B 0,C 180,E1 7940.028,E2 7940.028} C_VEL
LIN {X 0,Y 451.131,Z 691.44,A -85,B 0,C 180,E1 7945.859,E2 7945.859} C_VEL
LIN {X 0,Y 450.964,Z 691.44,A -85,B 0,C 180,E1 7952.482,E2 7952.482} C_VEL
LIN {X 0,Y 450.944,Z 691.44,A -85,B 0,C 180,E1 7957.171,E2 7957.171} C_VEL
LIN {X 0,Y 450.869,Z 691.44,A -85,B 0,C 180,E1 7962.179,E2 7962.179} C_VEL
LIN {X 0,Y 453.182,Z 696.998,A -85,B 0,C 180,E1 7962.633,E2 7962.633} C_VEL
LIN {X 0,Y 473.235,Z 731.52,A -85,B 0,C 180,E1 7966.195,E2 7966.195} C_VEL
LIN {X 0,Y 482.6,Z 752.937,A -85,B 0,C 180,E1 7968.161,E2 7968.161} C_VEL
LIN {X 0,Y 478.523,Z 793.029,A -85,B 0,C 180,E1 7970.04,E2 7970.04} C_VEL
LIN {X 0,Y 473.381,Z 830.956,A -85,B 0,C 180,E1 7972.576,E2 7972.576} C_VEL
LIN {X 0,Y 467.73,Z 867.566,A -85,B 0,C 180,E1 7975.936,E2 7975.936} C_VEL
LIN {X 0,Y 462.515,Z 899.355,A -85,B 0,C 180,E1 7979.804,E2 7979.804} C_VEL
LIN {X 0,Y 457.976,Z 929.268,A -85,B 0,C 180,E1 7984.546,E2 7984.546} C_VEL
LIN {X 0,Y 454.774,Z 953.066,A -85,B 0,C 180,E1 7989.55,E2 7989.55} C_VEL
LIN {X 0,Y 453.098,Z 971.516,A -85,B 0,C 180,E1 7994.859,E2 7994.859} C_VEL
LIN {X 0,Y 452.293,Z 984.414,A -85,B 0,C 180,E1 8000.364,E2 8000.364} C_VEL
LIN {X 0,Y 452.078,Z 989.953,A -85,B 0,C 180,E1 8004.233,E2 8004.233} C_VEL
LIN {X 0,Y 452.026,Z 992.671,A -85,B 0,C 180,E1 8008.08,E2 8008.08} C_VEL
LIN {X 0,Y 452.036,Z 992.638,A -85,B 0,C 180,E1 8011.919,E2 8011.919} C_VEL
LIN {X 0,Y 452.092,Z 988.646,A -85,B 0,C 180,E1 8016.731,E2 8016.731} C_VEL
LIN {X 0,Y 452.455,Z 980.329,A -85,B 0,C 180,E1 8021.582,E2 8021.582} C_VEL
LIN {X 0,Y 453.589,Z 965.543,A -85,B 0,C 180,E1 8026.982,E2 8026.982} C_VEL
LIN {X 0,Y 455.999,Z 943.972,A -85,B 0,C 180,E1 8032.447,E2 8032.447} C_VEL
LIN {X 0,Y 459.777,Z 917.099,A -85,B 0,C 180,E1 8037.453,E2 8037.453} C_VEL
LIN {X 0,Y 464.777,Z 885.1,A -85,B 0,C 180,E1 8041.972,E2 8041.972} C_VEL
LIN {X 0,Y 470.265,Z 851.178,A -85,B 0,C 180,E1 8045.609,E2 8045.609} C_VEL
LIN {X 0,Y 475.945,Z 813.045,A -85,B 0,C 180,E1 8048.64,E2 8048.64} C_VEL
LIN {X 0,Y 480.919,Z 772.203,A -85,B 0,C 180,E1 8050.938,E2 8050.938} C_VEL
LIN {X 0,Y 482.238,Z 751.798,A -85,B 0,C 180,E1 8051.841,E2 8051.841} C_VEL
LIN {X 0,Y 466.259,Z 718.421,A -85,B 0,C 180,E1 8054.998,E2 8054.998} C_VEL
LIN {X 0,Y 450.984,Z 692.315,A -85,B 0,C 180,E1 8057.688,E2 8057.688} C_VEL
LIN {X 0,Y 450.929,Z 691.44,A -85,B 0,C 180,E1 8057.827,E2 8057.827} C_VEL
LIN {X 0,Y 450.857,Z 691.44,A -85,B 0,C 180,E1 8063.704,E2 8063.704} C_VEL
LIN {X 0,Y 450.928,Z 691.44,A -85,B 0,C 180,E1 8069.768,E2 8069.768} C_VEL
LIN {X 0,Y 451.151,Z 691.44,A -85,B 0,C 180,E1 8076.26,E2 8076.26} C_VEL
LIN {X 0,Y 451.378,Z 691.44,A -85,B 0,C 180,E1 8082.436,E2 8082.436} C_VEL
LIN {X 0,Y 451.515,Z 691.44,A -85,B 0,C 180,E1 8088.399,E2 8088.399} C_VEL
LIN {X 0,Y 451.661,Z 691.44,A -85,B 0,C 180,E1 8094.234,E2 8094.234} C_VEL
LIN {X 0,Y 451.946,Z 691.44,A -85,B 0,C 180,E1 8100.005,E2 8100.005} C_VEL
LIN {X 0,Y 451.691,Z 691.44,A -85,B 0,C 180,E1 8105.775,E2 8105.775} C_VEL
LIN {X 0,Y 451.432,Z 691.44,A -85,B 0,C 180,E1 8111.612,E2 8111.612} C_VEL
LIN {X 0,Y 451.294,Z 691.44,A -85,B 0,C 180,E1 8117.577,E2 8117.577} C_VEL
LIN {X 0,Y 451.16,Z 691.44,A -85,B 0,C 180,E1 8123.75,E2 8123.75} C_VEL
LIN {X 0,Y 450.935,Z 691.44,A -85,B 0,C 180,E1 8130.242,E2 8130.242} C_VEL
LIN {X 0,Y 450.894,Z 691.44,A -85,B 0,C 180,E1 8137.188,E2 8137.188} C_VEL
LIN {X 0,Y 450.959,Z 691.44,A -85,B 0,C 180,E1 8141.709,E2 8141.709} C_VEL
LIN {X 0,Y 453.182,Z 696.948,A -85,B 0,C 180,E1 8142.154,E2 8142.154} C_VEL
LIN {X 0,Y 473.698,Z 731.064,A -85,B 0,C 180,E1 8145.53,E2 8145.53} C_VEL
LIN {X 0,Y 484.529,Z 752.361,A -85,B 0,C 180,E1 8147.336,E2 8147.336} C_VEL
LIN {X 0,Y 481.109,Z 792.996,A -85,B 0,C 180,E1 8148.696,E2 8148.696} C_VEL
LIN {X 0,Y 477.632,Z 825.084,A -85,B 0,C 180,E1 8150.307,E2 8150.307} C_VEL
LIN {X 0,Y 472.428,Z 840.908,A -85,B 0,C 180,E1 8150.982,E2 8150.982} C_VEL
LIN {X 0,Y 467.422,Z 854.365,A -85,B 0,C 180,E1 8151.646,E2 8151.646} C_VEL
LIN {X 0,Y 467.086,Z 856.226,A -85,B 0,C 180,E1 8151.781,E2 8151.781} C_VEL
LIN {X 0,Y 461.009,Z 894.466,A -85,B 0,C 180,E1 8155.189,E2 8155.189} C_VEL
LIN {X 0,Y 455.447,Z 928.602,A -85,B 0,C 180,E1 8159.263,E2 8159.263} C_VEL
LIN {X 0,Y 450.758,Z 958.017,A -85,B 0,C 180,E1 8163.904,E2 8163.904} C_VEL
LIN {X 0,Y 447.288,Z 982.129,A -85,B 0,C 180,E1 8168.992,E2 8168.992} C_VEL
LIN {X 0,Y 445.352,Z 1000.293,A -85,B 0,C 180,E1 8174.218,E2 8174.218} C_VEL
LIN {X 0,Y 444.46,Z 1012.406,A -85,B 0,C 180,E1 8179.202,E2 8179.202} C_VEL
LIN {X 0,Y 444.214,Z 1019.905,A -85,B 0,C 180,E1 8184.131,E2 8184.131} C_VEL
LIN {X 0,Y 444.199,Z 1022.657,A -85,B 0,C 180,E1 8188.047,E2 8188.047} C_VEL
LIN {X 0,Y 444.085,Z 1022.657,A -85,B 0,C 180,E1 8191.954,E2 8191.954} C_VEL
LIN {X 0,Y 444.259,Z 1018.703,A -85,B 0,C 180,E1 8196.851,E2 8196.851} C_VEL
LIN {X 0,Y 444.595,Z 1010.433,A -85,B 0,C 180,E1 8201.791,E2 8201.791} C_VEL
LIN {X 0,Y 445.788,Z 995.684,A -85,B 0,C 180,E1 8207.289,E2 8207.289} C_VEL
LIN {X 0,Y 448.363,Z 974.173,A -85,B 0,C 180,E1 8212.852,E2 8212.852} C_VEL
LIN {X 0,Y 452.434,Z 947.361,A -85,B 0,C 180,E1 8217.938,E2 8217.938} C_VEL
LIN {X 0,Y 457.506,Z 915.942,A -85,B 0,C 180,E1 8222.377,E2 8222.377} C_VEL
LIN {X 0,Y 463.344,Z 880.54,A -85,B 0,C 180,E1 8226.167,E2 8226.167} C_VEL
LIN {X 0,Y 469.15,Z 842.048,A -85,B 0,C 180,E1 8229.238,E2 8229.238} C_VEL
LIN {X 0,Y 474.485,Z 800.555,A -85,B 0,C 180,E1 8231.583,E2 8231.583} C_VEL
LIN {X 0,Y 478.04,Z 762.929,A -85,B 0,C 180,E1 8232.995,E2 8232.995} C_VEL
LIN {X 0,Y 477.985,Z 754.312,A -85,B 0,C 180,E1 8233.319,E2 8233.319} C_VEL
LIN {X 0,Y 458.505,Z 717.901,A -85,B 0,C 180,E1 8236.659,E2 8236.659} C_VEL
LIN {X 0,Y 443.28,Z 693.172,A -85,B 0,C 180,E1 8239.363,E2 8239.363} C_VEL
LIN {X 0,Y 443.074,Z 691.44,A -85,B 0,C 180,E1 8239.514,E2 8239.514} C_VEL
LIN {X 0,Y 442.962,Z 691.44,A -85,B 0,C 180,E1 8246.845,E2 8246.845} C_VEL
LIN {X 0,Y 443.128,Z 691.44,A -85,B 0,C 180,E1 8253.627,E2 8253.627} C_VEL
LIN {X 0,Y 443.362,Z 691.44,A -85,B 0,C 180,E1 8260.03,E2 8260.03} C_VEL
LIN {X 0,Y 443.326,Z 691.44,A -85,B 0,C 180,E1 8266.165,E2 8266.165} C_VEL
LIN {X 0,Y 443.684,Z 691.44,A -85,B 0,C 180,E1 8272.151,E2 8272.151} C_VEL
LIN {X 0,Y 444.042,Z 691.44,A -85,B 0,C 180,E1 8278.042,E2 8278.042} C_VEL
LIN {X 0,Y 443.867,Z 691.44,A -85,B 0,C 180,E1 8283.907,E2 8283.907} C_VEL
LIN {X 0,Y 443.659,Z 691.44,A -85,B 0,C 180,E1 8289.819,E2 8289.819} C_VEL
LIN {X 0,Y 443.438,Z 691.44,A -85,B 0,C 180,E1 8295.845,E2 8295.845} C_VEL
LIN {X 0,Y 443.258,Z 691.44,A -85,B 0,C 180,E1 8302.062,E2 8302.062} C_VEL
LIN {X 0,Y 443.087,Z 691.44,A -85,B 0,C 180,E1 8308.571,E2 8308.571} C_VEL
LIN {X 0,Y 443.058,Z 691.44,A -85,B 0,C 180,E1 8315.506,E2 8315.506} C_VEL
LIN {X 0,Y 442.899,Z 691.89,A -85,B 0,C 180,E1 8321.031,E2 8321.031} C_VEL
LIN {X 0,Y 445.427,Z 697.239,A -85,B 0,C 180,E1 8321.535,E2 8321.535} C_VEL
LIN {X 0,Y 465.796,Z 731.789,A -85,B 0,C 180,E1 8325.306,E2 8325.306} C_VEL
LIN {X 0,Y 476.523,Z 755.429,A -85,B 0,C 180,E1 8327.608,E2 8327.608} C_VEL
LIN {X 0,Y 471.969,Z 796.626,A -85,B 0,C 180,E1 8329.605,E2 8329.605} C_VEL
LIN {X 0,Y 466.464,Z 834.578,A -85,B 0,C 180,E1 8332.245,E2 8332.245} C_VEL
LIN {X 0,Y 460.843,Z 868.941,A -85,B 0,C 180,E1 8335.491,E2 8335.491} C_VEL
LIN {X 0,Y 455.495,Z 899.513,A -85,B 0,C 180,E1 8339.266,E2 8339.266} C_VEL
LIN {X 0,Y 450.527,Z 929.262,A -85,B 0,C 180,E1 8344.094,E2 8344.094} C_VEL
LIN {X 0,Y 447.088,Z 953.374,A -85,B 0,C 180,E1 8349.264,E2 8349.264} C_VEL
LIN {X 0,Y 445.389,Z 970.429,A -85,B 0,C 180,E1 8354.219,E2 8354.219} C_VEL
LIN {X 0,Y 444.528,Z 982.492,A -85,B 0,C 180,E1 8359.202,E2 8359.202} C_VEL
LIN {X 0,Y 444.18,Z 989.952,A -85,B 0,C 180,E1 8364.13,E2 8364.13} C_VEL
LIN {X 0,Y 444.123,Z 992.671,A -85,B 0,C 180,E1 8368.046,E2 8368.046} C_VEL
LIN {X 0,Y 444.13,Z 992.639,A -85,B 0,C 180,E1 8371.953,E2 8371.953} C_VEL
LIN {X 0,Y 444.206,Z 988.647,A -85,B 0,C 180,E1 8376.851,E2 8376.851} C_VEL
LIN {X 0,Y 444.6,Z 980.331,A -85,B 0,C 180,E1 8381.79,E2 8381.79} C_VEL
LIN {X 0,Y 445.857,Z 965.546,A -85,B 0,C 180,E1 8387.286,E2 8387.286} C_VEL
LIN {X 0,Y 448.461,Z 943.974,A -85,B 0,C 180,E1 8392.846,E2 8392.846} C_VEL
LIN {X 0,Y 452.5,Z 917.133,A -85,B 0,C 180,E1 8397.933,E2 8397.933} C_VEL
LIN {X 0,Y 457.715,Z 886.466,A -85,B 0,C 180,E1 8402.383,E2 8402.383} C_VEL
LIN {X 0,Y 463.653,Z 851.853,A -85,B 0,C 180,E1 8406.159,E2 8406.159} C_VEL
LIN {X 0,Y 469.654,Z 813.62,A -85,B 0,C 180,E1 8409.235,E2 8409.235} C_VEL
LIN {X 0,Y 474.928,Z 772.521,A -85,B 0,C 180,E1 8411.568,E2 8411.568} C_VEL
LIN {X 0,Y 476.049,Z 754.593,A -85,B 0,C 180,E1 8412.394,E2 8412.394} C_VEL
LIN {X 0,Y 459.729,Z 720.358,A -85,B 0,C 180,E1 8415.764,E2 8415.764} C_VEL
LIN {X 0,Y 444.804,Z 696.545,A -85,B 0,C 180,E1 8418.477,E2 8418.477} C_VEL
LIN {X 0,Y 442.916,Z 691.44,A -85,B 0,C 180,E1 8419.005,E2 8419.005} C_VEL
LIN {X 0,Y 442.932,Z 691.44,A -85,B 0,C 180,E1 8425.124,E2 8425.124} C_VEL
LIN {X 0,Y 443.037,Z 691.44,A -85,B 0,C 180,E1 8431.425,E2 8431.425} C_VEL
LIN {X 0,Y 443.268,Z 691.44,A -85,B 0,C 180,E1 8437.939,E2 8437.939} C_VEL
LIN {X 0,Y 443.501,Z 691.44,A -85,B 0,C 180,E1 8444.157,E2 8444.157} C_VEL
LIN {X 0,Y 443.693,Z 691.44,A -85,B 0,C 180,E1 8450.182,E2 8450.182} C_VEL
LIN {X 0,Y 443.96,Z 691.44,A -85,B 0,C 180,E1 8456.094,E2 8456.094} C_VEL
LIN {X 0,Y 444.055,Z 691.44,A -85,B 0,C 180,E1 8461.958,E2 8461.958} C_VEL
LIN {X 0,Y 443.634,Z 691.44,A -85,B 0,C 180,E1 8468.215,E2 8468.215} C_VEL
LIN {X 0,Y 443.478,Z 691.44,A -85,B 0,C 180,E1 8473.83,E2 8473.83} C_VEL
LIN {X 0,Y 443.334,Z 691.44,A -85,B 0,C 180,E1 8479.972,E2 8479.972} C_VEL
LIN {X 0,Y 443.154,Z 691.44,A -85,B 0,C 180,E1 8486.371,E2 8486.371} C_VEL
LIN {X 0,Y 442.946,Z 691.44,A -85,B 0,C 180,E1 8493.156,E2 8493.156} C_VEL
LIN {X 0,Y 443.08,Z 691.48,A -85,B 0,C 180,E1 8500.572,E2 8500.572} C_VEL
LIN {X 0,Y 445.369,Z 696.986,A -85,B 0,C 180,E1 8501.044,E2 8501.044} C_VEL
LIN {X 0,Y 466.937,Z 732.504,A -85,B 0,C 180,E1 8504.755,E2 8504.755} C_VEL
LIN {X 0,Y 478.423,Z 756.502,A -85,B 0,C 180,E1 8506.798,E2 8506.798} C_VEL
LIN {X 0,Y 474.358,Z 800.78,A -85,B 0,C 180,E1 8508.416,E2 8508.416} C_VEL
LIN {X 0,Y 469.161,Z 842.018,A -85,B 0,C 180,E1 8510.76,E2 8510.76} C_VEL
LIN {X 0,Y 467.086,Z 856.226,A -85,B 0,C 180,E1 8511.781,E2 8511.781} C_VEL
LIN {X 0,Y 461.429,Z 871.139,A -85,B 0,C 180,E1 8512.691,E2 8512.691} C_VEL
LIN {X 0,Y 456.082,Z 883.773,A -85,B 0,C 180,E1 8513.56,E2 8513.56} C_VEL
LIN {X 0,Y 455.737,Z 885.459,A -85,B 0,C 180,E1 8513.725,E2 8513.725} C_VEL
LIN {X 0,Y 450.025,Z 918.574,A -85,B 0,C 180,E1 8517.432,E2 8517.432} C_VEL
LIN {X 0,Y 444.669,Z 949.94,A -85,B 0,C 180,E1 8522.045,E2 8522.045} C_VEL
LIN {X 0,Y 440.759,Z 975.322,A -85,B 0,C 180,E1 8526.999,E2 8526.999} C_VEL
LIN {X 0,Y 438.153,Z 995.688,A -85,B 0,C 180,E1 8532.401,E2 8532.401} C_VEL
LIN {X 0,Y 436.726,Z 1010.434,A -85,B 0,C 180,E1 8537.994,E2 8537.994} C_VEL
LIN {X 0,Y 436.342,Z 1018.703,A -85,B 0,C 180,E1 8543.025,E2 8543.025} C_VEL
LIN {X 0,Y 436.308,Z 1022.657,A -85,B 0,C 180,E1 8548.012,E2 8548.012} C_VEL
LIN {X 0,Y 436.206,Z 1022.657,A -85,B 0,C 180,E1 8551.99,E2 8551.99} C_VEL
LIN {X 0,Y 436.358,Z 1018.702,A -85,B 0,C 180,E1 8556.976,E2 8556.976} C_VEL
LIN {X 0,Y 436.741,Z 1010.433,A -85,B 0,C 180,E1 8562.006,E2 8562.006} C_VEL
LIN {X 0,Y 438.048,Z 995.684,A -85,B 0,C 180,E1 8567.604,E2 8567.604} C_VEL
LIN {X 0,Y 440.765,Z 974.171,A -85,B 0,C 180,E1 8573.269,E2 8573.269} C_VEL
LIN {X 0,Y 444.911,Z 948.582,A -85,B 0,C 180,E1 8578.191,E2 8578.191} C_VEL
LIN {X 0,Y 450.373,Z 916.669,A -85,B 0,C 180,E1 8582.815,E2 8582.815} C_VEL
LIN {X 0,Y 456.758,Z 879.881,A -85,B 0,C 180,E1 8586.81,E2 8586.81} C_VEL
LIN {X 0,Y 463.041,Z 840.694,A -85,B 0,C 180,E1 8589.942,E2 8589.942} C_VEL
LIN {X 0,Y 468.509,Z 800.279,A -85,B 0,C 180,E1 8592.234,E2 8592.234} C_VEL
LIN {X 0,Y 472.315,Z 762.226,A -85,B 0,C 180,E1 8593.663,E2 8593.663} C_VEL
LIN {X 0,Y 471.881,Z 757.048,A -85,B 0,C 180,E1 8593.92,E2 8593.92} C_VEL
LIN {X 0,Y 452.542,Z 720.531,A -85,B 0,C 180,E1 8597.397,E2 8597.397} C_VEL
LIN {X 0,Y 436.996,Z 696.608,A -85,B 0,C 180,E1 8600.238,E2 8600.238} C_VEL
LIN {X 0,Y 435,Z 691.44,A -85,B 0,C 180,E1 8600.813,E2 8600.813} C_VEL
LIN {X 0,Y 435.061,Z 691.44,A -85,B 0,C 180,E1 8606.642,E2 8606.642} C_VEL
LIN {X 0,Y 435.184,Z 691.44,A -85,B 0,C 180,E1 8613.108,E2 8613.108} C_VEL
LIN {X 0,Y 435.443,Z 691.44,A -85,B 0,C 180,E1 8619.855,E2 8619.855} C_VEL
LIN {X 0,Y 435.411,Z 691.44,A -85,B 0,C 180,E1 8626.823,E2 8626.823} C_VEL
LIN {X 0,Y 435.771,Z 691.44,A -85,B 0,C 180,E1 8632.007,E2 8632.007} C_VEL
LIN {X 0,Y 436.16,Z 691.44,A -85,B 0,C 180,E1 8638.006,E2 8638.006} C_VEL
LIN {X 0,Y 435.952,Z 691.44,A -85,B 0,C 180,E1 8643.978,E2 8643.978} C_VEL
LIN {X 0,Y 435.724,Z 691.44,A -85,B 0,C 180,E1 8649.999,E2 8649.999} C_VEL
LIN {X 0,Y 435.541,Z 691.44,A -85,B 0,C 180,E1 8656.14,E2 8656.14} C_VEL
LIN {X 0,Y 435.326,Z 691.44,A -85,B 0,C 180,E1 8662.485,E2 8662.485} C_VEL
LIN {X 0,Y 435.091,Z 691.44,A -85,B 0,C 180,E1 8669.543,E2 8669.543} C_VEL
LIN {X 0,Y 435.038,Z 691.44,A -85,B 0,C 180,E1 8676.263,E2 8676.263} C_VEL
LIN {X 0,Y 434.954,Z 691.798,A -85,B 0,C 180,E1 8679.801,E2 8679.801} C_VEL
LIN {X 0,Y 437.385,Z 697.09,A -85,B 0,C 180,E1 8680.317,E2 8680.317} C_VEL
LIN {X 0,Y 457.426,Z 730.219,A -85,B 0,C 180,E1 8684.186,E2 8684.186} C_VEL
LIN {X 0,Y 470.439,Z 759.096,A -85,B 0,C 180,E1 8687.092,E2 8687.092} C_VEL
LIN {X 0,Y 465.197,Z 802.259,A -85,B 0,C 180,E1 8689.282,E2 8689.282} C_VEL
LIN {X 0,Y 459.048,Z 841.658,A -85,B 0,C 180,E1 8692.198,E2 8692.198} C_VEL
LIN {X 0,Y 452.6,Z 877.905,A -85,B 0,C 180,E1 8695.886,E2 8695.886} C_VEL
LIN {X 0,Y 446.424,Z 910.686,A -85,B 0,C 180,E1 8700.368,E2 8700.368} C_VEL
LIN {X 0,Y 441.784,Z 937.829,A -85,B 0,C 180,E1 8705.326,E2 8705.326} C_VEL
LIN {X 0,Y 438.86,Z 958.863,A -85,B 0,C 180,E1 8710.343,E2 8710.343} C_VEL
LIN {X 0,Y 437.072,Z 975.883,A -85,B 0,C 180,E1 8715.966,E2 8715.966} C_VEL
LIN {X 0,Y 436.449,Z 985.86,A -85,B 0,C 180,E1 8720.937,E2 8720.937} C_VEL
LIN {X 0,Y 436.261,Z 991.657,A -85,B 0,C 180,E1 8726.019,E2 8726.019} C_VEL
LIN {X 0,Y 436.217,Z 992.998,A -85,B 0,C 180,E1 8730,E2 8730} C_VEL
LIN {X 0,Y 436.164,Z 991.594,A -85,B 0,C 180,E1 8733.981,E2 8733.981} C_VEL
LIN {X 0,Y 436.437,Z 985.737,A -85,B 0,C 180,E1 8739.053,E2 8739.053} C_VEL
LIN {X 0,Y 437.239,Z 974.446,A -85,B 0,C 180,E1 8744.488,E2 8744.488} C_VEL
LIN {X 0,Y 438.817,Z 958.536,A -85,B 0,C 180,E1 8749.658,E2 8749.658} C_VEL
LIN {X 0,Y 441.755,Z 937.458,A -85,B 0,C 180,E1 8754.669,E2 8754.669} C_VEL
LIN {X 0,Y 446.622,Z 909.981,A -85,B 0,C 180,E1 8759.652,E2 8759.652} C_VEL
LIN {X 0,Y 452.782,Z 877.169,A -85,B 0,C 180,E1 8764.106,E2 8764.106} C_VEL
LIN {X 0,Y 459.098,Z 841.802,A -85,B 0,C 180,E1 8767.691,E2 8767.691} C_VEL
LIN {X 0,Y 465.167,Z 802.463,A -85,B 0,C 180,E1 8770.615,E2 8770.615} C_VEL
LIN {X 0,Y 470.252,Z 758.483,A -85,B 0,C 180,E1 8772.869,E2 8772.869} C_VEL
LIN {X 0,Y 454.534,Z 724.93,A -85,B 0,C 180,E1 8776.289,E2 8776.289} C_VEL
LIN {X 0,Y 437.308,Z 697.034,A -85,B 0,C 180,E1 8779.599,E2 8779.599} C_VEL
LIN {X 0,Y 434.934,Z 691.44,A -85,B 0,C 180,E1 8780.196,E2 8780.196} C_VEL
LIN {X 0,Y 435.03,Z 691.44,A -85,B 0,C 180,E1 8786.646,E2 8786.646} C_VEL
LIN {X 0,Y 435.187,Z 691.44,A -85,B 0,C 180,E1 8793.119,E2 8793.119} C_VEL
LIN {X 0,Y 435.434,Z 691.44,A -85,B 0,C 180,E1 8799.856,E2 8799.856} C_VEL
LIN {X 0,Y 435.64,Z 691.44,A -85,B 0,C 180,E1 8806.691,E2 8806.691} C_VEL
LIN {X 0,Y 435.805,Z 691.44,A -85,B 0,C 180,E1 8812.018,E2 8812.018} C_VEL
LIN {X 0,Y 436.054,Z 691.44,A -85,B 0,C 180,E1 8818.015,E2 8818.015} C_VEL
LIN {X 0,Y 435.875,Z 691.44,A -85,B 0,C 180,E1 8823.988,E2 8823.988} C_VEL
LIN {X 0,Y 435.617,Z 691.44,A -85,B 0,C 180,E1 8830.012,E2 8830.012} C_VEL
LIN {X 0,Y 435.502,Z 691.44,A -85,B 0,C 180,E1 8836.151,E2 8836.151} C_VEL
LIN {X 0,Y 435.333,Z 691.44,A -85,B 0,C 180,E1 8842.495,E2 8842.495} C_VEL
LIN {X 0,Y 435.058,Z 691.44,A -85,B 0,C 180,E1 8849.159,E2 8849.159} C_VEL
LIN {X 0,Y 435.023,Z 691.44,A -85,B 0,C 180,E1 8853.84,E2 8853.84} C_VEL
LIN {X 0,Y 435.031,Z 691.524,A -85,B 0,C 180,E1 8859.332,E2 8859.332} C_VEL
LIN {X 0,Y 437.268,Z 696.924,A -85,B 0,C 180,E1 8859.82,E2 8859.82} C_VEL
LIN {X 0,Y 456.868,Z 728.035,A -85,B 0,C 180,E1 8863.364,E2 8863.364} C_VEL
LIN {X 0,Y 472.453,Z 758.376,A -85,B 0,C 180,E1 8866.199,E2 8866.199} C_VEL
LIN {X 0,Y 468.213,Z 801.747,A -85,B 0,C 180,E1 8867.826,E2 8867.826} C_VEL
LIN {X 0,Y 462.604,Z 843.6,A -85,B 0,C 180,E1 8870.255,E2 8870.255} C_VEL
LIN {X 0,Y 456.45,Z 881.546,A -85,B 0,C 180,E1 8873.34,E2 8873.34} C_VEL
LIN {X 0,Y 455.737,Z 885.459,A -85,B 0,C 180,E1 8873.725,E2 8873.725} C_VEL
LIN {X 0,Y 450.012,Z 899.368,A -85,B 0,C 180,E1 8874.889,E2 8874.889} C_VEL
LIN {X 0,Y 444.142,Z 912.578,A -85,B 0,C 180,E1 8876.145,E2 8876.145} C_VEL
LIN {X 0,Y 438.492,Z 942.924,A -85,B 0,C 180,E1 8880.426,E2 8880.426} C_VEL
LIN {X 0,Y 433.974,Z 969.166,A -85,B 0,C 180,E1 8885.25,E2 8885.25} C_VEL
LIN {X 0,Y 431.06,Z 988.702,A -85,B 0,C 180,E1 8889.973,E2 8889.973} C_VEL
LIN {X 0,Y 429.375,Z 1004.428,A -85,B 0,C 180,E1 8895.188,E2 8895.188} C_VEL
LIN {X 0,Y 428.645,Z 1014.33,A -85,B 0,C 180,E1 8899.828,E2 8899.828} C_VEL
LIN {X 0,Y 428.424,Z 1019.905,A -85,B 0,C 180,E1 8903.914,E2 8903.914} C_VEL
LIN {X 0,Y 428.4,Z 1022.657,A -85,B 0,C 180,E1 8907.975,E2 8907.975} C_VEL
LIN {X 0,Y 428.301,Z 1022.657,A -85,B 0,C 180,E1 8912.026,E2 8912.026} C_VEL
LIN {X 0,Y 428.468,Z 1018.702,A -85,B 0,C 180,E1 8917.105,E2 8917.105} C_VEL
LIN {X 0,Y 428.892,Z 1010.432,A -85,B 0,C 180,E1 8922.229,E2 8922.229} C_VEL
LIN {X 0,Y 430.235,Z 996.158,A -85,B 0,C 180,E1 8927.773,E2 8927.773} C_VEL
LIN {X 0,Y 432.921,Z 976.342,A -85,B 0,C 180,E1 8933.17,E2 8933.17} C_VEL
LIN {X 0,Y 436.961,Z 951.574,A -85,B 0,C 180,E1 8938.124,E2 8938.124} C_VEL
LIN {X 0,Y 442.379,Z 922.154,A -85,B 0,C 180,E1 8942.62,E2 8942.62} C_VEL
LIN {X 0,Y 448.501,Z 889.399,A -85,B 0,C 180,E1 8946.457,E2 8946.457} C_VEL
LIN {X 0,Y 454.761,Z 853.649,A -85,B 0,C 180,E1 8949.633,E2 8949.633} C_VEL
LIN {X 0,Y 460.694,Z 814.699,A -85,B 0,C 180,E1 8952.159,E2 8952.159} C_VEL
LIN {X 0,Y 465.363,Z 773.91,A -85,B 0,C 180,E1 8953.97,E2 8953.97} C_VEL
LIN {X 0,Y 466.028,Z 760.537,A -85,B 0,C 180,E1 8954.461,E2 8954.461} C_VEL
LIN {X 0,Y 448.237,Z 726.115,A -85,B 0,C 180,E1 8957.861,E2 8957.861} C_VEL
LIN {X 0,Y 429.598,Z 697.235,A -85,B 0,C 180,E1 8961.412,E2 8961.412} C_VEL
LIN {X 0,Y 427.152,Z 692.807,A -85,B 0,C 180,E1 8961.939,E2 8961.939} C_VEL
LIN {X 0,Y 427.01,Z 691.44,A -85,B 0,C 180,E1 8962.126,E2 8962.126} C_VEL
LIN {X 0,Y 427.127,Z 691.44,A -85,B 0,C 180,E1 8968.295,E2 8968.295} C_VEL
LIN {X 0,Y 427.31,Z 691.44,A -85,B 0,C 180,E1 8974.835,E2 8974.835} C_VEL
LIN {X 0,Y 427.491,Z 691.44,A -85,B 0,C 180,E1 8981.41,E2 8981.41} C_VEL
LIN {X 0,Y 427.547,Z 691.44,A -85,B 0,C 180,E1 8987.729,E2 8987.729} C_VEL
LIN {X 0,Y 427.93,Z 691.44,A -85,B 0,C 180,E1 8993.903,E2 8993.903} C_VEL
LIN {X 0,Y 428.183,Z 691.44,A -85,B 0,C 180,E1 8999.995,E2 8999.995} C_VEL
LIN {X 0,Y 427.908,Z 691.44,A -85,B 0,C 180,E1 9006.088,E2 9006.088} C_VEL
LIN {X 0,Y 427.679,Z 691.44,A -85,B 0,C 180,E1 9012.257,E2 9012.257} C_VEL
LIN {X 0,Y 427.536,Z 691.44,A -85,B 0,C 180,E1 9018.578,E2 9018.578} C_VEL
LIN {X 0,Y 427.322,Z 691.44,A -85,B 0,C 180,E1 9025.153,E2 9025.153} C_VEL
LIN {X 0,Y 427.171,Z 691.44,A -85,B 0,C 180,E1 9032.107,E2 9032.107} C_VEL
LIN {X 0,Y 427.031,Z 691.44,A -85,B 0,C 180,E1 9038.474,E2 9038.474} C_VEL
LIN {X 0,Y 429.358,Z 697.021,A -85,B 0,C 180,E1 9039.025,E2 9039.025} C_VEL
LIN {X 0,Y 447.386,Z 725.808,A -85,B 0,C 180,E1 9042.667,E2 9042.667} C_VEL
LIN {X 0,Y 463.108,Z 758.438,A -85,B 0,C 180,E1 9046.192,E2 9046.192} C_VEL
LIN {X 0,Y 464.217,Z 763.598,A -85,B 0,C 180,E1 9046.609,E2 9046.609} C_VEL
LIN {X 0,Y 458.755,Z 805.073,A -85,B 0,C 180,E1 9048.795,E2 9048.795} C_VEL
LIN {X 0,Y 452.29,Z 844.11,A -85,B 0,C 180,E1 9051.769,E2 9051.769} C_VEL
LIN {X 0,Y 445.642,Z 879.483,A -85,B 0,C 180,E1 9055.461,E2 9055.461} C_VEL
LIN {X 0,Y 439.49,Z 910.43,A -85,B 0,C 180,E1 9059.752,E2 9059.752} C_VEL
LIN {X 0,Y 434.555,Z 937.17,A -85,B 0,C 180,E1 9064.672,E2 9064.672} C_VEL
LIN {X 0,Y 430.965,Z 960.639,A -85,B 0,C 180,E1 9070.503,E2 9070.503} C_VEL
LIN {X 0,Y 429.248,Z 975.88,A -85,B 0,C 180,E1 9075.705,E2 9075.705} C_VEL
LIN {X 0,Y 428.586,Z 986.084,A -85,B 0,C 180,E1 9080.916,E2 9080.916} C_VEL
LIN {X 0,Y 428.354,Z 991.656,A -85,B 0,C 180,E1 9085.946,E2 9085.946} C_VEL
LIN {X 0,Y 428.317,Z 992.998,A -85,B 0,C 180,E1 9090,E2 9090} C_VEL
LIN {X 0,Y 428.26,Z 991.595,A -85,B 0,C 180,E1 9094.054,E2 9094.054} C_VEL
LIN {X 0,Y 428.547,Z 985.819,A -85,B 0,C 180,E1 9099.168,E2 9099.168} C_VEL
LIN {X 0,Y 429.31,Z 975.649,A -85,B 0,C 180,E1 9104.292,E2 9104.292} C_VEL
LIN {X 0,Y 430.949,Z 960.353,A -85,B 0,C 180,E1 9109.497,E2 9109.497} C_VEL
LIN {X 0,Y 434.569,Z 936.801,A -85,B 0,C 180,E1 9115.32,E2 9115.32} C_VEL
LIN {X 0,Y 439.662,Z 909.689,A -85,B 0,C 180,E1 9120.277,E2 9120.277} C_VEL
LIN {X 0,Y 446.214,Z 876.683,A -85,B 0,C 180,E1 9124.783,E2 9124.783} C_VEL
LIN {X 0,Y 452.745,Z 842.113,A -85,B 0,C 180,E1 9128.315,E2 9128.315} C_VEL
LIN {X 0,Y 459.162,Z 802.772,A -85,B 0,C 180,E1 9131.261,E2 9131.261} C_VEL
LIN {X 0,Y 464.193,Z 761.602,A -85,B 0,C 180,E1 9133.419,E2 9133.419} C_VEL
LIN {X 0,Y 449.637,Z 729.944,A -85,B 0,C 180,E1 9136.775,E2 9136.775} C_VEL
LIN {X 0,Y 433.031,Z 702.592,A -85,B 0,C 180,E1 9140.133,E2 9140.133} C_VEL
LIN {X 0,Y 427.165,Z 692.873,A -85,B 0,C 180,E1 9141.352,E2 9141.352} C_VEL
LIN {X 0,Y 427.002,Z 691.44,A -85,B 0,C 180,E1 9141.603,E2 9141.603} C_VEL
LIN {X 0,Y 427.119,Z 691.44,A -85,B 0,C 180,E1 9148.295,E2 9148.295} C_VEL
LIN {X 0,Y 427.321,Z 691.44,A -85,B 0,C 180,E1 9154.847,E2 9154.847} C_VEL
LIN {X 0,Y 427.558,Z 691.44,A -85,B 0,C 180,E1 9161.423,E2 9161.423} C_VEL
LIN {X 0,Y 427.767,Z 691.44,A -85,B 0,C 180,E1 9167.745,E2 9167.745} C_VEL
LIN {X 0,Y 427.914,Z 691.44,A -85,B 0,C 180,E1 9173.912,E2 9173.912} C_VEL
LIN {X 0,Y 428.25,Z 691.44,A -85,B 0,C 180,E1 9180.005,E2 9180.005} C_VEL
LIN {X 0,Y 427.937,Z 691.44,A -85,B 0,C 180,E1 9186.097,E2 9186.097} C_VEL
LIN {X 0,Y 427.662,Z 691.44,A -85,B 0,C 180,E1 9192.268,E2 9192.268} C_VEL
LIN {X 0,Y 427.491,Z 691.44,A -85,B 0,C 180,E1 9198.59,E2 9198.59} C_VEL
LIN {X 0,Y 427.335,Z 691.44,A -85,B 0,C 180,E1 9205.163,E2 9205.163} C_VEL
LIN {X 0,Y 427.093,Z 691.44,A -85,B 0,C 180,E1 9212.125,E2 9212.125} C_VEL
LIN {X 0,Y 427.011,Z 691.44,A -85,B 0,C 180,E1 9218.008,E2 9218.008} C_VEL
LIN {X 0,Y 429.363,Z 697.002,A -85,B 0,C 180,E1 9218.553,E2 9218.553} C_VEL
LIN {X 0,Y 446.68,Z 723.735,A -85,B 0,C 180,E1 9221.866,E2 9221.866} C_VEL
LIN {X 0,Y 463.767,Z 755.74,A -85,B 0,C 180,E1 9225.074,E2 9225.074} C_VEL
LIN {X 0,Y 466.386,Z 761.923,A -85,B 0,C 180,E1 9225.638,E2 9225.638} C_VEL
LIN {X 0,Y 462.192,Z 802.021,A -85,B 0,C 180,E1 9227.184,E2 9227.184} C_VEL
LIN {X 0,Y 456.346,Z 843.401,A -85,B 0,C 180,E1 9229.608,E2 9229.608} C_VEL
LIN {X 0,Y 449.672,Z 882.421,A -85,B 0,C 180,E1 9232.833,E2 9232.833} C_VEL
LIN {X 0,Y 444.142,Z 912.578,A -85,B 0,C 180,E1 9236.145,E2 9236.145} C_VEL
LIN {X 0,Y 438.312,Z 925.259,A -85,B 0,C 180,E1 9237.525,E2 9237.525} C_VEL
LIN {X 0,Y 432.413,Z 937.262,A -85,B 0,C 180,E1 9239.019,E2 9239.019} C_VEL
LIN {X 0,Y 426.966,Z 966.405,A -85,B 0,C 180,E1 9244.253,E2 9244.253} C_VEL
LIN {X 0,Y 423.408,Z 988.602,A -85,B 0,C 180,E1 9249.595,E2 9249.595} C_VEL
LIN {X 0,Y 421.586,Z 1004.427,A -85,B 0,C 180,E1 9254.908,E2 9254.908} C_VEL
LIN {X 0,Y 420.758,Z 1014.33,A -85,B 0,C 180,E1 9259.635,E2 9259.635} C_VEL
LIN {X 0,Y 420.523,Z 1019.905,A -85,B 0,C 180,E1 9263.8,E2 9263.8} C_VEL
LIN {X 0,Y 420.493,Z 1022.657,A -85,B 0,C 180,E1 9267.937,E2 9267.937} C_VEL
LIN {X 0,Y 420.397,Z 1022.657,A -85,B 0,C 180,E1 9272.064,E2 9272.064} C_VEL
LIN {X 0,Y 420.597,Z 1018.702,A -85,B 0,C 180,E1 9277.239,E2 9277.239} C_VEL
LIN {X 0,Y 421.028,Z 1010.432,A -85,B 0,C 180,E1 9282.461,E2 9282.461} C_VEL
LIN {X 0,Y 422.633,Z 995.224,A -85,B 0,C 180,E1 9288.418,E2 9288.418} C_VEL
LIN {X 0,Y 425.713,Z 973.755,A -85,B 0,C 180,E1 9294.143,E2 9294.143} C_VEL
LIN {X 0,Y 430.624,Z 946.436,A -85,B 0,C 180,E1 9299.489,E2 9299.489} C_VEL
LIN {X 0,Y 436.81,Z 914.897,A -85,B 0,C 180,E1 9304.132,E2 9304.132} C_VEL
LIN {X 0,Y 443.677,Z 879.606,A -85,B 0,C 180,E1 9308.047,E2 9308.047} C_VEL
LIN {X 0,Y 450.621,Z 840.71,A -85,B 0,C 180,E1 9311.226,E2 9311.226} C_VEL
LIN {X 0,Y 456.787,Z 798.882,A -85,B 0,C 180,E1 9313.63,E2 9313.63} C_VEL
LIN {X 0,Y 460.137,Z 763.821,A -85,B 0,C 180,E1 9315.035,E2 9315.035} C_VEL
LIN {X 0,Y 443.203,Z 730.559,A -85,B 0,C 180,E1 9318.452,E2 9318.452} C_VEL
LIN {X 0,Y 425.6,Z 703.093,A -85,B 0,C 180,E1 9321.93,E2 9321.93} C_VEL
LIN {X 0,Y 421.023,Z 696.545,A -85,B 0,C 180,E1 9322.905,E2 9322.905} C_VEL
LIN {X 0,Y 419.072,Z 691.44,A -85,B 0,C 180,E1 9323.581,E2 9323.581} C_VEL
LIN {X 0,Y 419.243,Z 691.44,A -85,B 0,C 180,E1 9330.084,E2 9330.084} C_VEL
LIN {X 0,Y 419.4,Z 691.44,A -85,B 0,C 180,E1 9336.6,E2 9336.6} C_VEL
LIN {X 0,Y 419.566,Z 691.44,A -85,B 0,C 180,E1 9343.217,E2 9343.217} C_VEL
LIN {X 0,Y 419.716,Z 691.44,A -85,B 0,C 180,E1 9349.605,E2 9349.605} C_VEL
LIN {X 0,Y 420.063,Z 691.44,A -85,B 0,C 180,E1 9355.862,E2 9355.862} C_VEL
LIN {X 0,Y 420.194,Z 691.44,A -85,B 0,C 180,E1 9362.06,E2 9362.06} C_VEL
LIN {X 0,Y 419.958,Z 691.44,A -85,B 0,C 180,E1 9368.285,E2 9368.285} C_VEL
LIN {X 0,Y 419.711,Z 691.44,A -85,B 0,C 180,E1 9374.619,E2 9374.619} C_VEL
LIN {X 0,Y 419.512,Z 691.44,A -85,B 0,C 180,E1 9381.148,E2 9381.148} C_VEL
LIN {X 0,Y 419.284,Z 691.44,A -85,B 0,C 180,E1 9387.988,E2 9387.988} C_VEL
LIN {X 0,Y 419.194,Z 691.44,A -85,B 0,C 180,E1 9395.291,E2 9395.291} C_VEL
LIN {X 0,Y 419.19,Z 691.44,A -85,B 0,C 180,E1 9397.078,E2 9397.078} C_VEL
LIN {X 0,Y 421.33,Z 696.916,A -85,B 0,C 180,E1 9397.643,E2 9397.643} C_VEL
LIN {X 0,Y 437.588,Z 722.002,A -85,B 0,C 180,E1 9401.09,E2 9401.09} C_VEL
LIN {X 0,Y 454.286,Z 754.909,A -85,B 0,C 180,E1 9404.909,E2 9404.909} C_VEL
LIN {X 0,Y 458.308,Z 765.464,A -85,B 0,C 180,E1 9406,E2 9406} C_VEL
LIN {X 0,Y 452.701,Z 805.833,A -85,B 0,C 180,E1 9408.161,E2 9408.161} C_VEL
LIN {X 0,Y 446.079,Z 843.979,A -85,B 0,C 180,E1 9411.09,E2 9411.09} C_VEL
LIN {X 0,Y 438.963,Z 879.781,A -85,B 0,C 180,E1 9414.859,E2 9414.859} C_VEL
LIN {X 0,Y 432.265,Z 911.69,A -85,B 0,C 180,E1 9419.37,E2 9419.37} C_VEL
LIN {X 0,Y 427.149,Z 937.735,A -85,B 0,C 180,E1 9424.264,E2 9424.264} C_VEL
LIN {X 0,Y 423.467,Z 958.985,A -85,B 0,C 180,E1 9429.598,E2 9429.598} C_VEL
LIN {X 0,Y 421.46,Z 975.877,A -85,B 0,C 180,E1 9435.435,E2 9435.435} C_VEL
LIN {X 0,Y 420.695,Z 985.985,A -85,B 0,C 180,E1 9440.679,E2 9440.679} C_VEL
LIN {X 0,Y 420.46,Z 991.656,A -85,B 0,C 180,E1 9445.87,E2 9445.87} C_VEL
LIN {X 0,Y 420.417,Z 992.998,A -85,B 0,C 180,E1 9450,E2 9450} C_VEL
LIN {X 0,Y 420.375,Z 991.595,A -85,B 0,C 180,E1 9454.13,E2 9454.13} C_VEL
LIN {X 0,Y 420.66,Z 985.851,A -85,B 0,C 180,E1 9459.321,E2 9459.321} C_VEL
LIN {X 0,Y 421.486,Z 975.651,A -85,B 0,C 180,E1 9464.563,E2 9464.563} C_VEL
LIN {X 0,Y 423.451,Z 958.681,A -85,B 0,C 180,E1 9470.402,E2 9470.402} C_VEL
LIN {X 0,Y 427.382,Z 936.078,A -85,B 0,C 180,E1 9476.002,E2 9476.002} C_VEL
LIN {X 0,Y 432.951,Z 908.475,A -85,B 0,C 180,E1 9481.057,E2 9481.057} C_VEL
LIN {X 0,Y 439.564,Z 876.999,A -85,B 0,C 180,E1 9485.387,E2 9485.387} C_VEL
LIN {X 0,Y 446.62,Z 841.684,A -85,B 0,C 180,E1 9489.018,E2 9489.018} C_VEL
LIN {X 0,Y 453.389,Z 801.841,A -85,B 0,C 180,E1 9492.001,E2 9492.001} C_VEL
LIN {X 0,Y 457.912,Z 764.274,A -85,B 0,C 180,E1 9494.028,E2 9494.028} C_VEL
LIN {X 0,Y 444.232,Z 733.928,A -85,B 0,C 180,E1 9497.373,E2 9497.373} C_VEL
LIN {X 0,Y 426.328,Z 703.916,A -85,B 0,C 180,E1 9501.201,E2 9501.201} C_VEL
LIN {X 0,Y 419.254,Z 693.103,A -85,B 0,C 180,E1 9502.733,E2 9502.733} C_VEL
LIN {X 0,Y 419.098,Z 691.44,A -85,B 0,C 180,E1 9503.01,E2 9503.01} C_VEL
LIN {X 0,Y 419.243,Z 691.44,A -85,B 0,C 180,E1 9510.083,E2 9510.083} C_VEL
LIN {X 0,Y 419.415,Z 691.44,A -85,B 0,C 180,E1 9516.612,E2 9516.612} C_VEL
LIN {X 0,Y 419.739,Z 691.44,A -85,B 0,C 180,E1 9523.235,E2 9523.235} C_VEL
LIN {X 0,Y 419.904,Z 691.44,A -85,B 0,C 180,E1 9529.62,E2 9529.62} C_VEL
LIN {X 0,Y 420.201,Z 691.44,A -85,B 0,C 180,E1 9535.873,E2 9535.873} C_VEL
LIN {X 0,Y 420.341,Z 691.44,A -85,B 0,C 180,E1 9542.069,E2 9542.069} C_VEL
LIN {X 0,Y 419.943,Z 691.44,A -85,B 0,C 180,E1 9548.296,E2 9548.296} C_VEL
LIN {X 0,Y 419.696,Z 691.44,A -85,B 0,C 180,E1 9554.63,E2 9554.63} C_VEL
LIN {X 0,Y 419.496,Z 691.44,A -85,B 0,C 180,E1 9561.16,E2 9561.16} C_VEL
LIN {X 0,Y 419.266,Z 691.44,A -85,B 0,C 180,E1 9568.001,E2 9568.001} C_VEL
LIN {X 0,Y 419.102,Z 691.44,A -85,B 0,C 180,E1 9575.313,E2 9575.313} C_VEL
LIN {X 0,Y 419.105,Z 691.892,A -85,B 0,C 180,E1 9576.634,E2 9576.634} C_VEL
LIN {X 0,Y 421.697,Z 697.258,A -85,B 0,C 180,E1 9577.247,E2 9577.247} C_VEL
LIN {X 0,Y 439.659,Z 724.65,A -85,B 0,C 180,E1 9580.867,E2 9580.867} C_VEL
LIN {X 0,Y 456.596,Z 756.041,A -85,B 0,C 180,E1 9584.197,E2 9584.197} C_VEL
LIN {X 0,Y 460.362,Z 765.539,A -85,B 0,C 180,E1 9585.066,E2 9585.066} C_VEL
LIN {X 0,Y 455.882,Z 805.051,A -85,B 0,C 180,E1 9586.668,E2 9586.668} C_VEL
LIN {X 0,Y 450.047,Z 843.734,A -85,B 0,C 180,E1 9588.982,E2 9588.982} C_VEL
LIN {X 0,Y 443.141,Z 882.218,A -85,B 0,C 180,E1 9592.203,E2 9592.203} C_VEL
LIN {X 0,Y 436.227,Z 917.957,A -85,B 0,C 180,E1 9596.267,E2 9596.267} C_VEL
LIN {X 0,Y 432.413,Z 937.262,A -85,B 0,C 180,E1 9599.019,E2 9599.019} C_VEL
LIN {X 0,Y 426.558,Z 948.581,A -85,B 0,C 180,E1 9600.631,E2 9600.631} C_VEL
LIN {X 0,Y 420.837,Z 959.159,A -85,B 0,C 180,E1 9602.36,E2 9602.36} C_VEL
LIN {X 0,Y 416.731,Z 982.623,A -85,B 0,C 180,E1 9607.659,E2 9607.659} C_VEL
LIN {X 0,Y 414.276,Z 1000.166,A -85,B 0,C 180,E1 9613,E2 9613} C_VEL
LIN {X 0,Y 413.028,Z 1012.405,A -85,B 0,C 180,E1 9618.369,E2 9618.369} C_VEL
LIN {X 0,Y 412.624,Z 1019.905,A -85,B 0,C 180,E1 9623.68,E2 9623.68} C_VEL
LIN {X 0,Y 412.586,Z 1022.657,A -85,B 0,C 180,E1 9627.897,E2 9627.897} C_VEL
LIN {X 0,Y 412.492,Z 1022.657,A -85,B 0,C 180,E1 9632.104,E2 9632.104} C_VEL
LIN {X 0,Y 412.711,Z 1018.092,A -85,B 0,C 180,E1 9637.913,E2 9637.913} C_VEL
LIN {X 0,Y 413.31,Z 1008.921,A -85,B 0,C 180,E1 9643.407,E2 9643.407} C_VEL
LIN {X 0,Y 414.85,Z 995.292,A -85,B 0,C 180,E1 9648.675,E2 9648.675} C_VEL
LIN {X 0,Y 418.096,Z 974.187,A -85,B 0,C 180,E1 9654.436,E2 9654.436} C_VEL
LIN {X 0,Y 423.246,Z 947.175,A -85,B 0,C 180,E1 9659.864,E2 9659.864} C_VEL
LIN {X 0,Y 430.017,Z 914.653,A -85,B 0,C 180,E1 9664.739,E2 9664.739} C_VEL
LIN {X 0,Y 437.255,Z 879.301,A -85,B 0,C 180,E1 9668.709,E2 9668.709} C_VEL
LIN {X 0,Y 444.452,Z 841.049,A -85,B 0,C 180,E1 9671.871,E2 9671.871} C_VEL
LIN {X 0,Y 450.929,Z 799.232,A -85,B 0,C 180,E1 9674.305,E2 9674.305} C_VEL
LIN {X 0,Y 454.156,Z 766.924,A -85,B 0,C 180,E1 9675.649,E2 9675.649} C_VEL
LIN {X 0,Y 438.308,Z 735.138,A -85,B 0,C 180,E1 9679.039,E2 9679.039} C_VEL
LIN {X 0,Y 420.973,Z 707.824,A -85,B 0,C 180,E1 9682.604,E2 9682.604} C_VEL
LIN {X 0,Y 413.731,Z 697.26,A -85,B 0,C 180,E1 9684.229,E2 9684.229} C_VEL
LIN {X 0,Y 411.28,Z 692.593,A -85,B 0,C 180,E1 9684.839,E2 9684.839} C_VEL
LIN {X 0,Y 411.19,Z 691.44,A -85,B 0,C 180,E1 9685.072,E2 9685.072} C_VEL
LIN {X 0,Y 411.361,Z 691.44,A -85,B 0,C 180,E1 9692.051,E2 9692.051} C_VEL
LIN {X 0,Y 411.535,Z 691.44,A -85,B 0,C 180,E1 9698.411,E2 9698.411} C_VEL
LIN {X 0,Y 411.602,Z 691.44,A -85,B 0,C 180,E1 9705.075,E2 9705.075} C_VEL
LIN {X 0,Y 411.994,Z 691.44,A -85,B 0,C 180,E1 9711.543,E2 9711.543} C_VEL
LIN {X 0,Y 412.417,Z 691.44,A -85,B 0,C 180,E1 9717.891,E2 9717.891} C_VEL
LIN {X 0,Y 412.21,Z 691.44,A -85,B 0,C 180,E1 9724.207,E2 9724.207} C_VEL
LIN {X 0,Y 411.918,Z 691.44,A -85,B 0,C 180,E1 9730.584,E2 9730.584} C_VEL
LIN {X 0,Y 411.741,Z 691.44,A -85,B 0,C 180,E1 9737.101,E2 9737.101} C_VEL
LIN {X 0,Y 411.456,Z 691.44,A -85,B 0,C 180,E1 9743.868,E2 9743.868} C_VEL
LIN {X 0,Y 411.354,Z 691.44,A -85,B 0,C 180,E1 9748.577,E2 9748.577} C_VEL
LIN {X 0,Y 411.305,Z 692.029,A -85,B 0,C 180,E1 9755.632,E2 9755.632} C_VEL
LIN {X 0,Y 413.929,Z 697.384,A -85,B 0,C 180,E1 9756.295,E2 9756.295} C_VEL
LIN {X 0,Y 430.702,Z 723.163,A -85,B 0,C 180,E1 9760.059,E2 9760.059} C_VEL
LIN {X 0,Y 447.51,Z 756.123,A -85,B 0,C 180,E1 9764.078,E2 9764.078} C_VEL
LIN {X 0,Y 452.237,Z 769.194,A -85,B 0,C 180,E1 9765.461,E2 9765.461} C_VEL
LIN {X 0,Y 446.299,Z 808.897,A -85,B 0,C 180,E1 9767.663,E2 9767.663} C_VEL
LIN {X 0,Y 439.421,Z 846.251,A -85,B 0,C 180,E1 9770.616,E2 9770.616} C_VEL
LIN {X 0,Y 432.098,Z 881.115,A -85,B 0,C 180,E1 9774.37,E2 9774.37} C_VEL
LIN {X 0,Y 425.236,Z 912.124,A -85,B 0,C 180,E1 9778.833,E2 9778.833} C_VEL
LIN {X 0,Y 419.554,Z 939.215,A -85,B 0,C 180,E1 9784.051,E2 9784.051} C_VEL
LIN {X 0,Y 415.859,Z 959.286,A -85,B 0,C 180,E1 9789.207,E2 9789.207} C_VEL
LIN {X 0,Y 413.645,Z 975.897,A -85,B 0,C 180,E1 9795.153,E2 9795.153} C_VEL
LIN {X 0,Y 412.825,Z 985.984,A -85,B 0,C 180,E1 9800.5,E2 9800.5} C_VEL
LIN {X 0,Y 412.552,Z 991.655,A -85,B 0,C 180,E1 9805.79,E2 9805.79} C_VEL
LIN {X 0,Y 412.517,Z 992.998,A -85,B 0,C 180,E1 9810,E2 9810} C_VEL
LIN {X 0,Y 412.47,Z 991.596,A -85,B 0,C 180,E1 9814.21,E2 9814.21} C_VEL
LIN {X 0,Y 412.799,Z 985.853,A -85,B 0,C 180,E1 9819.5,E2 9819.5} C_VEL
LIN {X 0,Y 413.656,Z 975.681,A -85,B 0,C 180,E1 9824.845,E2 9824.845} C_VEL
LIN {X 0,Y 415.576,Z 960.76,A -85,B 0,C 180,E1 9830.25,E2 9830.25} C_VEL
LIN {X 0,Y 419.326,Z 940.031,A -85,B 0,C 180,E1 9835.676,E2 9835.676} C_VEL
LIN {X 0,Y 424.774,Z 914.218,A -85,B 0,C 180,E1 9840.718,E2 9840.718} C_VEL
LIN {X 0,Y 431.35,Z 884.655,A -85,B 0,C 180,E1 9845.084,E2 9845.084} C_VEL
LIN {X 0,Y 438.359,Z 851.688,A -85,B 0,C 180,E1 9848.776,E2 9848.776} C_VEL
LIN {X 0,Y 445.517,Z 813.892,A -85,B 0,C 180,E1 9851.902,E2 9851.902} C_VEL
LIN {X 0,Y 451.659,Z 773.373,A -85,B 0,C 180,E1 9854.266,E2 9854.266} C_VEL
LIN {X 0,Y 451.838,Z 767.336,A -85,B 0,C 180,E1 9854.611,E2 9854.611} C_VEL
LIN {X 0,Y 438.117,Z 736.458,A -85,B 0,C 180,E1 9858.145,E2 9858.145} C_VEL
LIN {X 0,Y 421.675,Z 709.024,A -85,B 0,C 180,E1 9861.84,E2 9861.84} C_VEL
LIN {X 0,Y 413.703,Z 697.276,A -85,B 0,C 180,E1 9863.646,E2 9863.646} C_VEL
LIN {X 0,Y 411.232,Z 692.536,A -85,B 0,C 180,E1 9864.261,E2 9864.261} C_VEL
LIN {X 0,Y 411.182,Z 691.44,A -85,B 0,C 180,E1 9864.444,E2 9864.444} C_VEL
LIN {X 0,Y 411.354,Z 691.44,A -85,B 0,C 180,E1 9872.052,E2 9872.052} C_VEL
LIN {X 0,Y 411.547,Z 691.44,A -85,B 0,C 180,E1 9878.422,E2 9878.422} C_VEL
LIN {X 0,Y 411.846,Z 691.44,A -85,B 0,C 180,E1 9885.095,E2 9885.095} C_VEL
LIN {X 0,Y 412.057,Z 691.44,A -85,B 0,C 180,E1 9891.554,E2 9891.554} C_VEL
LIN {X 0,Y 412.336,Z 691.44,A -85,B 0,C 180,E1 9897.901,E2 9897.901} C_VEL
LIN {X 0,Y 412.15,Z 691.44,A -85,B 0,C 180,E1 9904.218,E2 9904.218} C_VEL
LIN {X 0,Y 411.843,Z 691.44,A -85,B 0,C 180,E1 9910.596,E2 9910.596} C_VEL
LIN {X 0,Y 411.711,Z 691.44,A -85,B 0,C 180,E1 9917.113,E2 9917.113} C_VEL
LIN {X 0,Y 411.468,Z 691.44,A -85,B 0,C 180,E1 9923.879,E2 9923.879} C_VEL
LIN {X 0,Y 411.332,Z 691.44,A -85,B 0,C 180,E1 9928.59,E2 9928.59} C_VEL
LIN {X 0,Y 411.188,Z 691.44,A -85,B 0,C 180,E1 9935.121,E2 9935.121} C_VEL
LIN {X 0,Y 413.461,Z 697.006,A -85,B 0,C 180,E1 9935.728,E2 9935.728} C_VEL
LIN {X 0,Y 416.729,Z 701.717,A -85,B 0,C 180,E1 9936.475,E2 9936.475} C_VEL
LIN {X 0,Y 434.263,Z 728.197,A -85,B 0,C 180,E1 9940.151,E2 9940.151} C_VEL
LIN {X 0,Y 451.043,Z 759.908,A -85,B 0,C 180,E1 9943.649,E2 9943.649} C_VEL
LIN {X 0,Y 454.436,Z 768.628,A -85,B 0,C 180,E1 9944.461,E2 9944.461} C_VEL
LIN {X 0,Y 449.385,Z 810.028,A -85,B 0,C 180,E1 9946.243,E2 9946.243} C_VEL
LIN {X 0,Y 442.989,Z 848.95,A -85,B 0,C 180,E1 9948.709,E2 9948.709} C_VEL
LIN {X 0,Y 435.893,Z 885.747,A -85,B 0,C 180,E1 9951.936,E2 9951.936} C_VEL
LIN {X 0,Y 429.046,Z 919.178,A -85,B 0,C 180,E1 9955.864,E2 9955.864} C_VEL
LIN {X 0,Y 422.642,Z 950.016,A -85,B 0,C 180,E1 9960.648,E2 9960.648} C_VEL
LIN {X 0,Y 420.837,Z 959.159,A -85,B 0,C 180,E1 9962.36,E2 9962.36} C_VEL
LIN {X 0,Y 415.205,Z 969.028,A -85,B 0,C 180,E1 9964.2,E2 9964.2} C_VEL
LIN {X 0,Y 409.877,Z 978.091,A -85,B 0,C 180,E1 9966.142,E2 9966.142} C_VEL
LIN {X 0,Y 406.811,Z 997.845,A -85,B 0,C 180,E1 9971.959,E2 9971.959} C_VEL
LIN {X 0,Y 405.264,Z 1011.306,A -85,B 0,C 180,E1 9977.595,E2 9977.595} C_VEL
LIN {X 0,Y 404.798,Z 1018.418,A -85,B 0,C 180,E1 9982.224,E2 9982.224} C_VEL
LIN {X 0,Y 404.688,Z 1022.657,A -85,B 0,C 180,E1 9987.856,E2 9987.856} C_VEL
LIN {X 0,Y 404.601,Z 1022.657,A -85,B 0,C 180,E1 9992.145,E2 9992.145} C_VEL
LIN {X 0,Y 404.793,Z 1018.404,A -85,B 0,C 180,E1 9997.789,E2 9997.789} C_VEL
LIN {X 0,Y 405.336,Z 1010.265,A -85,B 0,C 180,E1 10002.952,E2 10002.952} C_VEL
LIN {X 0,Y 406.969,Z 995.956,A -85,B 0,C 180,E1 10008.707,E2 10008.707} C_VEL
LIN {X 0,Y 410.222,Z 975.922,A -85,B 0,C 180,E1 10014.401,E2 10014.401} C_VEL
LIN {X 0,Y 415.335,Z 950.263,A -85,B 0,C 180,E1 10019.807,E2 10019.807} C_VEL
LIN {X 0,Y 421.852,Z 920.567,A -85,B 0,C 180,E1 10024.528,E2 10024.528} C_VEL
LIN {X 0,Y 429.014,Z 888.003,A -85,B 0,C 180,E1 10028.465,E2 10028.465} C_VEL
LIN {X 0,Y 436.447,Z 851.225,A -85,B 0,C 180,E1 10031.801,E2 10031.801} C_VEL
LIN {X 0,Y 443.303,Z 812.308,A -85,B 0,C 180,E1 10034.337,E2 10034.337} C_VEL
LIN {X 0,Y 448.49,Z 773.164,A -85,B 0,C 180,E1 10036.081,E2 10036.081} C_VEL
LIN {X 0,Y 447.353,Z 767.816,A -85,B 0,C 180,E1 10036.493,E2 10036.493} C_VEL
LIN {X 0,Y 431.591,Z 736.441,A -85,B 0,C 180,E1 10040.027,E2 10040.027} C_VEL
LIN {X 0,Y 414.376,Z 709.498,A -85,B 0,C 180,E1 10043.755,E2 10043.755} C_VEL
LIN {X 0,Y 405.95,Z 697.366,A -85,B 0,C 180,E1 10045.765,E2 10045.765} C_VEL
LIN {X 0,Y 403.357,Z 692.418,A -85,B 0,C 180,E1 10046.46,E2 10046.46} C_VEL
LIN {X 0,Y 403.278,Z 691.44,A -85,B 0,C 180,E1 10046.814,E2 10046.814} C_VEL
LIN {X 0,Y 403.413,Z 691.44,A -85,B 0,C 180,E1 10053.23,E2 10053.23} C_VEL
LIN {X 0,Y 403.659,Z 691.44,A -85,B 0,C 180,E1 10060.268,E2 10060.268} C_VEL
LIN {X 0,Y 403.768,Z 691.44,A -85,B 0,C 180,E1 10067.156,E2 10067.156} C_VEL
LIN {X 0,Y 404.188,Z 691.44,A -85,B 0,C 180,E1 10073.543,E2 10073.543} C_VEL
LIN {X 0,Y 404.485,Z 691.44,A -85,B 0,C 180,E1 10079.995,E2 10079.995} C_VEL
LIN {X 0,Y 404.179,Z 691.44,A -85,B 0,C 180,E1 10086.447,E2 10086.447} C_VEL
LIN {X 0,Y 403.913,Z 691.44,A -85,B 0,C 180,E1 10092.991,E2 10092.991} C_VEL
LIN {X 0,Y 403.684,Z 691.44,A -85,B 0,C 180,E1 10099.72,E2 10099.72} C_VEL
LIN {X 0,Y 403.455,Z 691.44,A -85,B 0,C 180,E1 10106.755,E2 10106.755} C_VEL
LIN {X 0,Y 403.342,Z 691.445,A -85,B 0,C 180,E1 10113.989,E2 10113.989} C_VEL
LIN {X 0,Y 405.522,Z 696.882,A -85,B 0,C 180,E1 10114.615,E2 10114.615} C_VEL
LIN {X 0,Y 408.37,Z 700.644,A -85,B 0,C 180,E1 10115.308,E2 10115.308} C_VEL
LIN {X 0,Y 426.297,Z 728.57,A -85,B 0,C 180,E1 10119.562,E2 10119.562} C_VEL
LIN {X 0,Y 442.143,Z 760.555,A -85,B 0,C 180,E1 10123.583,E2 10123.583} C_VEL
LIN {X 0,Y 446.316,Z 771.184,A -85,B 0,C 180,E1 10124.814,E2 10124.814} C_VEL
LIN {X 0,Y 440.022,Z 811.283,A -85,B 0,C 180,E1 10127.101,E2 10127.101} C_VEL
LIN {X 0,Y 432.928,Z 847.946,A -85,B 0,C 180,E1 10130.073,E2 10130.073} C_VEL
LIN {X 0,Y 425.54,Z 881.413,A -85,B 0,C 180,E1 10133.734,E2 10133.734} C_VEL
LIN {X 0,Y 418.279,Z 912.425,A -85,B 0,C 180,E1 10138.255,E2 10138.255} C_VEL
LIN {X 0,Y 412.214,Z 939.518,A -85,B 0,C 180,E1 10143.553,E2 10143.553} C_VEL
LIN {X 0,Y 408.251,Z 959.589,A -85,B 0,C 180,E1 10148.801,E2 10148.801} C_VEL
LIN {X 0,Y 405.873,Z 976.197,A -85,B 0,C 180,E1 10154.862,E2 10154.862} C_VEL
LIN {X 0,Y 404.952,Z 986.032,A -85,B 0,C 180,E1 10160.313,E2 10160.313} C_VEL
LIN {X 0,Y 404.663,Z 991.654,A -85,B 0,C 180,E1 10165.708,E2 10165.708} C_VEL
LIN {X 0,Y 404.616,Z 992.998,A -85,B 0,C 180,E1 10170,E2 10170} C_VEL
LIN {X 0,Y 404.587,Z 991.597,A -85,B 0,C 180,E1 10174.292,E2 10174.292} C_VEL
LIN {X 0,Y 404.93,Z 985.908,A -85,B 0,C 180,E1 10179.686,E2 10179.686} C_VEL
